# B&R Automation Studio project NAINV104C00R8L515F00 (part 28)

#### Act_Background_RequestedBoardChk.st
```iecst
(** 2023-04-11 **)
ACTION Act_Background_RequestedBoardChk:

	IF eStatus2 <> Error  THEN
		bBoardChkReq := FALSE;
		memset(ADR(tyBoardAvailableReq),0,SIZEOF(tyBoardAvailableReq));
		IF bProcessBoardForecastId AND bNotAvlNotRdy  THEN //process boardforecast
			tyBoardAvailableReq.tyAvl.bProductTypeId	 		:= tyBoardForecastAcc.tyAvl.bProductTypeId;
			tyBoardAvailableReq.tyData.sProductTypeId 			:= tyBoardForecastAcc.tyData.sProductTypeId	;
			tyBoardAvailableReq.tyAvl.bThickness 				:= tyBoardForecastAcc.tyAvl.bThickness;
			tyBoardAvailableReq.tyAvl.bWidth 					:= tyBoardForecastAcc.tyAvl.bWidth;
			tyBoardAvailableReq.tyData.rWidth 					:= tyBoardForecastAcc.tyData.rWidth;
			tyBoardAvailableReq.tyAvl.bTopClearanceHeight 		:= tyBoardForecastAcc.tyAvl.bTopClearanceHeight;
			tyBoardAvailableReq.tyAvl.bBottomClearanceHeight 	:= tyBoardForecastAcc.tyAvl.bBottomClearanceHeight;
			tyBoardAvailableReq.tyData.eFlippedBoard 			:= tyBoardForecastAcc.tyData.eFlippedBoard;
			tyBoardAvailableReq.tyData.rThickness 				:= tyBoardForecastAcc.tyData.rThickness;
			tyBoardAvailableReq.tyData.rTopClearanceHeight 		:= tyBoardForecastAcc.tyData.rTopClearanceHeight;
			tyBoardAvailableReq.tyData.rBottomClearanceHeight 	:= tyBoardForecastAcc.tyData.rBottomClearanceHeight;
			bBoardChkReq := TRUE;
		ELSIF  bRcvBoardInfoOk AND bManuallInsertLastZone THEN //process query board info
			tyBoardAvailableReq.tyAvl.bProductTypeId	 		:= tySendBoardInfoAcc.tyAvl.bProductTypeId;
			tyBoardAvailableReq.tyData.sProductTypeId 			:= tySendBoardInfoAcc.tyData.sProductTypeId;
			tyBoardAvailableReq.tyAvl.bThickness 				:= tySendBoardInfoAcc.tyAvl.bThickness;
			tyBoardAvailableReq.tyAvl.bWidth 					:= tySendBoardInfoAcc.tyAvl.bWidth;
			tyBoardAvailableReq.tyData.rWidth 					:= tySendBoardInfoAcc.tyData.rWidth;
			tyBoardAvailableReq.tyAvl.bTopClearanceHeight 		:= tySendBoardInfoAcc.tyAvl.bTopClearanceHeight;
			tyBoardAvailableReq.tyAvl.bBottomClearanceHeight 	:= tySendBoardInfoAcc.tyAvl.bBottomClearanceHeight;
			tyBoardAvailableReq.tyData.eFlippedBoard 			:= tySendBoardInfoAcc.tyData.eFlippedBoard;
			tyBoardAvailableReq.tyData.rThickness 				:= tySendBoardInfoAcc.tyData.rThickness;
			tyBoardAvailableReq.tyData.rTopClearanceHeight 		:= tySendBoardInfoAcc.tyData.rTopClearanceHeight;
			tyBoardAvailableReq.tyData.rBottomClearanceHeight 	:= tySendBoardInfoAcc.tyData.rBottomClearanceHeight;
			bBoardChkReq := TRUE;
		ELSIF p_bAccDataRdy THEN
			memcpy(ADR(tyBoardAvailableReq),ADR(tyBoardAvailableRcv),SIZEOF(tyBoardAvailableRcv));
			bBoardChkReq := TRUE;
		END_IF
		//ADD
		IF bBoardChkReq AND (bTransporting = FALSE) AND (p_bOpsRun = TRUE) THEN

			bAccDataReq		:= FALSE;
			bBABlkUS		:= FALSE;
			bOverWriteSlt	:= FALSE;
			bOverWriteWidth	:= FALSE;

			IF p_tyParam.bCmpTypeId = TRUE THEN	//"Compare Type ID" Ticked

				IF tyBoardAvailableReq.tyAvl.bProductTypeId = TRUE THEN	//Check if there is Product Type Id in B.A msg

					IF tyBoardAvailableReq.tyData.sProductTypeId <> p_sRecipeNm THEN	//Product Type Id Different

						bAccDataReq	    := TRUE;	//Require To Load New Recipe
						bBABlkUS		:= TRUE;

						sReqRecipeNm	:= tyBoardAvailableReq.tyData.sProductTypeId;
						diReqWidthInUM	:= REAL_TO_DINT(tyBoardAvailableReq.tyData.rWidth * 1000);

					ELSE	//Product Type Id Same (After accepted or Originally same)

						IF p_tyParam.bCmpParam = TRUE THEN	//"Compare Param" Ticked
							IF tyBoardAvailableReq.tyAvl.bThickness AND tyBoardAvailableReq.tyAvl.bTopClearanceHeight AND tyBoardAvailableReq.tyAvl.bBottomClearanceHeight AND p_bBASltEn THEN	//Camparing Slot Parameters if p_bBASltEn = TRUE
								udiStatus2	:= fHermesCmpSlt(tyBoardAvailableReq.tyData.eFlippedBoard , tyBoardAvailableReq.tyData.rThickness , tyBoardAvailableReq.tyData.rTopClearanceHeight , tyBoardAvailableReq.tyData.rBottomClearanceHeight , p_diMinSltValue , p_diMaxSltValue , p_diPitch , p_diSltToSltInUM , p_diTtlSlt);

								IF udiStatus2 <> 0 THEN

									bBABlkUS	:= TRUE;

									eStatus2	:= Error;

									IF udiStatus2 = 2914 THEN
										udiStatus2	:= 10108;	//Input First Slot Is Invalid
									ELSIF udiStatus2 = 2915 THEN
										udiStatus2	:= 10109;	//Input Last Slot Is Invalid
									ELSIF udiStatus2 = 2916 THEN
										udiStatus2	:= 10110;	//Input Pitch Is Invalid
									ELSIF udiStatus2 = 2917 THEN
										udiStatus2	:= 10111;	//Input Slot To Slot Distance Is Invalid
									ELSIF udiStatus2 = 2918 THEN
										udiStatus2	:= 10112;	//Input Total Slot Is Invalid
									ELSIF udiStatus2 = 2919 THEN
										udiStatus2	:= 10113;	//Input Thickness Is Invalid
									ELSIF udiStatus2 = 2920 THEN
										udiStatus2	:= 10114;	//Input Top Clearance Height Is Invalid
									ELSIF udiStatus2 = 2921 THEN
										udiStatus2	:= 10115;	//Input Bottom Clearance Height Is Invalid
									ELSIF udiStatus2 = 2922 THEN
										udiStatus2	:= 10116;	//Recipe First Slot Value & Board Available Data Not Match With Same Product Type Id
									ELSIF udiStatus2 = 2923 THEN
										udiStatus2	:= 10117;	//Recipe Last Slot Value & Board Available Data Not Match With Same Product Type Id
									ELSIF udiStatus2 = 2924 THEN
										udiStatus2	:= 10118;	//Recipe Pitch Value & Board Available Data Not Match With Same Product Type Id
									END_IF

									fHermesAddOneMsgSend(ADR(a_eMsgSend) , ADR(udiMsgSendBffr) , HermesMsgTypeNotification);

									tyNotificationSnd.tyAvl.bSeverity			:= TRUE;
									tyNotificationSnd.tyAvl.bNotificationCode	:= TRUE;
									tyNotificationSnd.tyAvl.bDescription		:= TRUE;
									tyNotificationSnd.tyData.eSeverity			:= HermesSeverityError;
									tyNotificationSnd.tyData.iNotificationCode	:= UDINT_TO_INT(udiStatus2);
									tyNotificationSnd.tyData.sDescription		:= a_tyAlmText[udiStatus2].sAlmText;

								END_IF
							END_IF

							IF tyBoardAvailableReq.tyAvl.bWidth AND p_bBAWidthEn THEN	//Comparing Width Parameter if p_bBAWidthEn = TRUE
								IF REAL_TO_DINT(tyBoardAvailableReq.tyData.rWidth * 1000) <> p_diWidthInUM THEN

									bBABlkUS	:= TRUE;

									eStatus2	:= Error;
									udiStatus2	:= 10119;	//Width Different With Same Product Type Id

									fHermesAddOneMsgSend(ADR(a_eMsgSend) , ADR(udiMsgSendBffr) , HermesMsgTypeNotification);

									tyNotificationSnd.tyAvl.bSeverity			:= TRUE;
									tyNotificationSnd.tyAvl.bNotificationCode	:= TRUE;
									tyNotificationSnd.tyAvl.bDescription		:= TRUE;
									tyNotificationSnd.tyData.eSeverity			:= HermesSeverityError;
									tyNotificationSnd.tyData.iNotificationCode	:= UDINT_TO_INT(udiStatus2);
									tyNotificationSnd.tyData.sDescription		:= a_tyAlmText[udiStatus2].sAlmText;

								END_IF
							END_IF

						END_IF

					END_IF

				ELSE

					eStatus2	:= Error;
					udiStatus2	:= 10158;	//Product Type Id Not Receive From Upstream

					fHermesAddOneMsgSend(ADR(a_eMsgSend) , ADR(udiMsgSendBffr) , HermesMsgTypeNotification);

					tyNotificationSnd.tyAvl.bSeverity			:= TRUE;
					tyNotificationSnd.tyAvl.bNotificationCode	:= TRUE;
					tyNotificationSnd.tyAvl.bDescription		:= TRUE;
					tyNotificationSnd.tyData.eSeverity			:= HermesSeverityError;
					tyNotificationSnd.tyData.iNotificationCode	:= UDINT_TO_INT(udiStatus2);
					tyNotificationSnd.tyData.sDescription		:= a_tyAlmText[udiStatus2].sAlmText;

				END_IF

			ELSE	//"Compare Type ID" Not Ticked

				IF p_tyParam.bOverwrite THEN	//"Overwrite" Ticked

					IF tyBoardAvailableReq.tyAvl.bThickness AND tyBoardAvailableReq.tyAvl.bTopClearanceHeight AND tyBoardAvailableReq.tyAvl.bBottomClearanceHeight AND p_bBASltEn THEN	//Camparing Slot Parameters

						udiStatus2	:= fHermesCmpSlt(tyBoardAvailableReq.tyData.eFlippedBoard , tyBoardAvailableReq.tyData.rThickness , tyBoardAvailableReq.tyData.rTopClearanceHeight , tyBoardAvailableReq.tyData.rBottomClearanceHeight , p_diMinSltValue , p_diMaxSltValue , p_diPitch , p_diSltToSltInUM , p_diTtlSlt);

						IF udiStatus2 <> 0 THEN

							bAccDataReq		:= TRUE;
							bBABlkUS			:= TRUE;
							bOverWriteSlt	:= TRUE;

							fbGetSlt.eFlippedBrd				:= tyBoardAvailableReq.tyData.eFlippedBoard;
							fbGetSlt.rThicknessInMM				:= tyBoardAvailableReq.tyData.rThickness;
							fbGetSlt.rTopClearanceHeightInMM	:= tyBoardAvailableReq.tyData.rTopClearanceHeight;
							fbGetSlt.rBtmClearanceHeightInMM	:= tyBoardAvailableReq.tyData.rBottomClearanceHeight;
							fbGetSlt.diSltToSltInUM				:= p_diSltToSltInUM;
							fbGetSlt.diTtlSlt					:= p_diTtlSlt;
							fbGetSlt;

							diReqMinSltValue	:= fbGetSlt.diMinSltValue;
							diReqMaxSltValue	:= fbGetSlt.diMaxSltValue;
							diReqPitch			:= fbGetSlt.diPitch;

						END_IF

					END_IF

					IF tyBoardAvailableReq.tyAvl.bWidth  AND p_bBAWidthEn (*AND p_usiLinkProdRcpCurrRcpMcMod = 0*) THEN	//Comparing Width Parameter
						IF REAL_TO_DINT(tyBoardAvailableReq.tyData.rWidth * 1000) <> p_diWidthInUM THEN

							bAccDataReq		:= TRUE;
							bBABlkUS			:= TRUE;
							bOverWriteWidth	:= TRUE;

							diReqWidthInUM	:= REAL_TO_DINT(tyBoardAvailableReq.tyData.rWidth * 1000);

						END_IF
					END_IF

				ELSE	//"Compare Type ID" Not Ticked and "Overwrite" Not Ticked, Error if not same

					IF tyBoardAvailableReq.tyAvl.bThickness AND tyBoardAvailableReq.tyAvl.bTopClearanceHeight AND tyBoardAvailableReq.tyAvl.bBottomClearanceHeight AND p_bBASltEn AND p_bRdyRcv THEN	//Camparing Slot Parameters
						udiStatus2	:= fHermesCmpSlt(tyBoardAvailableReq.tyData.eFlippedBoard , tyBoardAvailableReq.tyData.rThickness , tyBoardAvailableReq.tyData.rTopClearanceHeight , tyBoardAvailableReq.tyData.rBottomClearanceHeight , p_diMinSltValue , p_diMaxSltValue , p_diPitch , p_diSltToSltInUM , p_diTtlSlt);

						IF udiStatus2 <> 0 THEN

							bBABlkUS		:= TRUE;

							eStatus2	:= Error;

							IF udiStatus2 = 2914 THEN
								udiStatus2	:= 10120;	//Input First Slot Is Invalid
							ELSIF udiStatus2 = 2915 THEN
								udiStatus2	:= 10121;	//Input Last Slot Is Invalid
							ELSIF udiStatus2 = 2916 THEN
								udiStatus2	:= 10122;	//Input Pitch Is Invalid
							ELSIF udiStatus2 = 2917 THEN
								udiStatus2	:= 10123;	//Input Slot To Slot Distance Is Invalid
							ELSIF udiStatus2 = 2918 THEN
								udiStatus2	:= 10124;	//Input Total Slot Is Invalid
							ELSIF udiStatus2 = 2919 THEN
								udiStatus2	:= 10125;	//Input Thickness Is Invalid
							ELSIF udiStatus2 = 2920 THEN
								udiStatus2	:= 10126;	//Input Top Clearance Height Is Invalid
							ELSIF udiStatus2 = 2921 THEN
								udiStatus2	:= 10127;	//Input Bottom Clearance Height Is Invalid
							ELSIF udiStatus2 = 2922 THEN
								udiStatus2	:= 10128;	//Recipe First Slot Value & Board Available Data Not Match With Same Product Type Id
							ELSIF udiStatus2 = 2923 THEN
								udiStatus2	:= 10129;	//Recipe Last Slot Value & Board Available Data Not Match With Same Product Type Id
							ELSIF udiStatus2 = 2924 THEN
								udiStatus2	:= 10130;	//Recipe Pitch Value & Board Available Data Not Match With Same Product Type Id
							END_IF

							fHermesAddOneMsgSend(ADR(a_eMsgSend) , ADR(udiMsgSendBffr) , HermesMsgTypeNotification);

							tyNotificationSnd.tyAvl.bSeverity			:= TRUE;
							tyNotificationSnd.tyAvl.bNotificationCode	:= TRUE;
							tyNotificationSnd.tyAvl.bDescription		:= TRUE;
							tyNotificationSnd.tyData.eSeverity			:= HermesSeverityError;
							tyNotificationSnd.tyData.iNotificationCode	:= UDINT_TO_INT(udiStatus2);
							tyNotificationSnd.tyData.sDescription		:= a_tyAlmText[udiStatus2].sAlmText;

						END_IF
					END_IF

					IF tyBoardAvailableReq.tyAvl.bWidth AND p_bBAWidthEn AND p_bRdyRcv THEN	//Comparing Width Parameter
						IF REAL_TO_DINT(tyBoardAvailableReq.tyData.rWidth * 1000) <> p_diWidthInUM THEN

							bBABlkUS		:= TRUE;

							eStatus2	:= Error;
							udiStatus2	:= 10131;	//Width Different With Same Product Type Id

							fHermesAddOneMsgSend(ADR(a_eMsgSend) , ADR(udiMsgSendBffr) , HermesMsgTypeNotification);

							tyNotificationSnd.tyAvl.bSeverity			:= TRUE;
							tyNotificationSnd.tyAvl.bNotificationCode	:= TRUE;
							tyNotificationSnd.tyAvl.bDescription		:= TRUE;
							tyNotificationSnd.tyData.eSeverity			:= HermesSeverityError;
							tyNotificationSnd.tyData.iNotificationCode	:= UDINT_TO_INT(udiStatus2);
							tyNotificationSnd.tyData.sDescription		:= a_tyAlmText[udiStatus2].sAlmText;

						END_IF
					END_IF

				END_IF

			END_IF
			                                                       //Add
		ELSIF NOT(bBoardChkReq) OR bTransporting = TRUE THEN //AND p_bUIInsertBrdPrep = FALSE THEN

			bAccDataReq		:= FALSE;
			bBABlkUS		:= FALSE;
			bOverWriteSlt	:= FALSE;
			bOverWriteWidth	:= FALSE;

		END_IF

		//reset bProcessBoardForecastId
		IF bProcessBoardForecastId = TRUE AND bBoardChkReq AND (bTransporting = FALSE) AND (p_bOpsRun = TRUE) THEN //reset condition
			IF bBABlkUS = FALSE OR  (bBFBlkUS AND eStatus2 = Error) THEN
				IF eStatus2 <> Error THEN
					bReplyMcRdyId := TRUE;
				END_IF
				bProcessBoardForecastId := FALSE;
			END_IF
		END_IF

	ELSE

		bAccDataReq		:= FALSE;
		bBABlkUS		:= TRUE;
		bOverWriteSlt	:= FALSE;
		bOverWriteWidth	:= FALSE;
		bBoardChkReq  := FALSE;
	END_IF

END_ACTION
```

#### Act_Background_Route.st
```iecst
(** 2021-08-01 **)
ACTION Act_Background_Route:

	//US Routing function

	//iGotoLane 0 Default Lane
	//iGotoLane 1 Route1
	IF NOT(p_bProcessRouteEn) THEN
		bReverseDSSndBfWBrdID := FALSE;
		bManualRmvBrdCond := FALSE;
		iGotoLane	:= 0;
		bProcessRouteReversal := FALSE;
		bTriggerRouteReversal := FALSE;
	ELSE
		// reversal condition
		IF EDGEPOS(tyBoardAvailableRcv.tyData.iRoute  = 900 AND tyBoardAvailableRcv.tyAvl.bRoute) THEN //flipping station reversal condition
			tyBoardAvailableRcv.tyAvl.bRoute := FALSE;
			bProcessRouteReversal := TRUE;
		ELSIF EDGEPOS(tyBoardAvailableRcv.tyAvl.bFlippedBoard  AND tyBoardAvailableRcv.tyData.eFlippedBoard = HermesFlippedBoardTopSideUp) THEN
			bTriggerRouteReversal := TRUE;
		END_IF

		//receiving Route
		IF	NOT(tyBoardAvailableRcv.tyAvl.bRoute)   THEN
			iGotoLane := 0; //default, depend on priority
		ELSE
			IF  p_bManualRmvRoute AND tyBoardAvailableRcv.tyData.iRoute  = 999  THEN
				bManualRmvBrdCond := TRUE;

			ELSIF p_bReturnRoute AND (
				(bProcessRouteReversal AND bProcessRouteMachine
				OR
				bTriggerRouteReversal AND bTriggerRouteMachine)
				OR bReverseDSSndBfWBrdID) THEN
				IF bProcessRouteReversal  THEN //Route Guide (900),flipper as downstream
					bReverseDSSndBfWBrdID := TRUE;
					bTriggerUpdateRoute  := FALSE;
					bProcessRouteReversal := FALSE;
				ELSIF bTriggerRouteReversal THEN //process as downstream
					bReverseDSSndBfWBrdID := TRUE;
					bTriggerUpdateRoute  := TRUE;
					bTriggerRouteReversal := FALSE;
				END_IF

				//Reset
				fbRstReverseDSSndBF(IN:= bReverseDSSndBfWBrdID AND NOT(p_bReceiveReverseUSMcRdy));
				IF (bReverseDSSndBfWBrdID AND p_bReceiveReverseUSMcRdy) OR fbRstReverseDSSndBF.Q THEN
					bReverseDSSndBfWBrdID := FALSE;
					bTriggerUpdateRoute := FALSE;
				END_IF
			ELSIF p_bNomRouteEn THEN
				iMinDis := 0;
				FOR usidx := 0 TO 2 DO
					//bChecking Closest Route
					IF tyBoardAvailableRcv.tyData.iRoute = pa_tyHermesDSParam[usidx].iLaneID THEN
						iGotoLane := usidx; //iGotoLane switch direction
						EXIT;
					ELSIF iMinDis = 0 THEN
						iMinDis := ABS(tyBoardAvailableRcv.tyData.iRoute - pa_tyHermesDSParam[usidx].iLaneID);
						iGotoLane := usidx;
					ELSE
						IF iMinDis > ABS(tyBoardAvailableRcv.tyData.iRoute - pa_tyHermesDSParam[usidx].iLaneID) THEN
							iGotoLane := usidx;
							iMinDis := ABS(tyBoardAvailableRcv.tyData.iRoute - pa_tyHermesDSParam[usidx].iLaneID);
						END_IF
					END_IF
				END_FOR
			END_IF
		END_IF

		//Process 900
		//when to reset block DS signal

		//Process 999
		//fbRstReverseDSSndBF(IN:= bManualRmvBrdCond);

	//	bBlkUS := bBlkUS OR bReverseDSSndBfWBrdID; //OR p_bSwitchtoReverseReceive;
	END_IF

	//reverse route, input receiving
	IF NOT(p_bReverseReceiveRoute) THEN
		bSwitchtoReverseReceive := FALSE;
	ELSE
		//process Reverse Input
		IF bSwitchtoReverseReceive = FALSE  AND EDGEPOS(p_tyDSHermesCurrBASnd.tyData.sBoardId = tyBoardForecastRcv.tyData.sBoardId AND tyBoardForecastRcv.tyData.sBoardId <> '' AND tyBoardForecastRcv.tyAvl.bBoardId) THEN
			tyBoardForecastRcv.tyAvl.bBoardId := FALSE;
			bSwitchtoReverseReceive := TRUE; //when to reset ReverseRcv back , if the BASnd not the same anymore
		ELSIF bSwitchtoReverseReceive = TRUE
			AND (EDGEPOS(tyMsgTypeRcv.bTransportFinished AND tyTransportFinished.tyData.eTransferState = HermesTransferStateComplete )
			OR EDGEPOS(tyMsgTypeRcv.bBoardForecast AND tyBoardForecastRcv.tyData.sBoardId = ''  )) THEN
			tyBoardForecastRcv.tyAvl.bBoardId := FALSE;
			bSwitchtoReverseReceive := FALSE;
		END_IF
		fbRstReverseRcvGate(IN:= bSwitchtoReverseReceive);
		bNotifyRstReverseRcvGate := fbRstReverseRcvGate.Q;
		//	bBlkUS := bBlkUS OR NOT(bSwitchtoReverseReceive);

		bReverseRcvBlkUS := NOT(bSwitchtoReverseReceive);
	END_IF

	//bBlkUS := bBlkUS OR p_bUSHermes2SwitchtoReverseRcv;
END_ACTION
```

#### Act_Background_Sequence.st
```iecst
 (** 2019-05-04 **)
ACTION Act_Background_Sequence:

	IF eStatus1 <> Error THEN

		IF p_bOpsRun = FALSE THEN
			p_bRcvIncompl	:= TRUE;
		END_IF

		IF tyMsgTypeRcv.bTransportFinished = TRUE THEN
			IF tyTransportFinished.tyData.eTransferState = HermesTransferStateNotStarted THEN
				p_bRcvNotStart	:= TRUE;
			ELSIF tyTransportFinished.tyData.eTransferState = HermesTransferStateIncomplete THEN
				p_bRcvIncompl	:= TRUE;
			END_IF
		END_IF

		bBlkUS := bBABlkUS OR  bBFBlkUS OR bManuallInsertLastZone
			OR bReverseDSSndBfWBrdID
			OR bReverseRcvBlkUS
			OR NOT(p_bHermesSwitchtoRvrseTransport); //no for reversal gate

		bBoardAvailableRcved := tyMsgTypeRcv.bBoardAvailable;

		//Sequence
		fbSequenceUS.bRstState		:= bRstState;
		fbSequenceUS.bRdyRcv		:= (p_bRdyRcv) AND (eStatus2 <> Error);
		fbSequenceUS.bBlkUS			:= bBlkUS;
		fbSequenceUS.bRdyTransport	:= p_bRdyTransport;
		fbSequenceUS.bRcvCompl		:= p_bRcvCompl;
		fbSequenceUS.bRcvIncompl	:= p_bRcvIncompl;
		fbSequenceUS.bRcvNotStart	:= p_bRcvNotStart;
		fbSequenceUS.bProcessBoardForecastId     	:= bProcessBoardForecastId; //Received BoardForecastId

		fbSequenceUS(bEn := TRUE);

		bNotAvlNotRdy                               := fbSequenceUS.bNotAvlNotRdy;

		bUSRdy		                               	:= fbSequenceUS.bUSRdy; //bUSRdy:= (eState = HermesStateBoardAvailable) OR (eState = HermesStateAvailableAndReady) OR (eState >= HermesStateTransporting);
		bDSRdy		                               	:= fbSequenceUS.bDSRdy;
		bTransporting                             	:= fbSequenceUS.bTransporting;
		bStopTransport                            	:= fbSequenceUS.bStopTransport;
		bUSGdRdy                                   	:= (tyBoardAvailableRcv.tyAvl.bFailedBoard = FALSE) OR ((tyBoardAvailableRcv.tyAvl.bFailedBoard = TRUE) AND (tyBoardAvailableRcv.tyData.eFailedBoard <> HermesFailedBoard));
		bDSGdRdy                                   	:= (tyMachineReady.tyAvl.bFailedBoard = FALSE) OR ((tyMachineReady.tyAvl.bFailedBoard = TRUE) AND (tyMachineReady.tyData.eFailedBoard <> HermesFailedBoard));

		//Action (defined 1 as bypass, 2 as flip)
		iAction										:= (tyBoardAvailableRcv.tyAvl.bAction = TRUE)*(tyBoardAvailableRcv.tyData.iAction);

		IF fbSequenceUS.eState >= HermesStateNotAvailableNotReady THEN
			bHandshakeDone	:= TRUE;
		ELSE
			bHandshakeDone	:= FALSE;
		END_IF

		IF EDGEPOS(fbSequenceUS.eState = HermesStateTransporting) THEN
			p_bRcvCompl		:= FALSE;
			p_bRcvIncompl	:= FALSE;
			p_bRcvNotStart	:= FALSE;
		END_IF

		IF fbSequenceUS.eMsgTypeSnd = HermesMsgTypeServiceDescription THEN
			fHermesAddOneMsgSend(ADR(a_eMsgSend) , ADR(udiMsgSendBffr) , HermesMsgTypeServiceDescription);

			tyServiceDescriptionSnd.tyData.sMachineId                                       := p_sMcId;
			tyServiceDescriptionSnd.tyData.iLaneId											:= p_tyParam.iLaneID;
			tyServiceDescriptionSnd.tyData.sInterfaceId										:= p_tyParam.sUpstreamInterfaceId;
			tyServiceDescriptionSnd.tyData.sVersion											:= p_sVersion;
			tyServiceDescriptionSnd.tyData.tySupportedFeatures.bFeatureCheckAliveResponse	:= (p_tyParam.bFeatureCheckAliveResponse) AND (p_tyParam.tRcvAlive <> T#0s) AND (p_tyParam.tSndAlive <> T#0s);
			tyServiceDescriptionSnd.tyData.tySupportedFeatures.bFeatureBoardForecast		:= p_tyParam.bFeatureBoardForecast;
			tyServiceDescriptionSnd.tyData.tySupportedFeatures.bFeatureQueryBoardInfo		:= p_tyParam.bFeatureQueryBoardInfo;
			tyServiceDescriptionSnd.tyData.tySupportedFeatures.bFeatureSendBoardInfo		:= FALSE;

			tyServiceDescriptionSnd.tyAvl.bMachineId										:= TRUE;
			tyServiceDescriptionSnd.tyAvl.bLaneId											:= tyServiceDescriptionSnd.tyData.iLaneId <> 0;
			tyServiceDescriptionSnd.tyAvl.bInterfaceId										:= tyServiceDescriptionSnd.tyData.sInterfaceId <> '';
			tyServiceDescriptionSnd.tyAvl.bVersion											:= TRUE;
			tyServiceDescriptionSnd.tyAvl.bSupportedFeatures								:= p_tyParam.bFeatureCheckAliveResponse OR p_tyParam.bFeatureBoardForecast OR p_tyParam.bFeatureQueryBoardInfo;
			tyServiceDescriptionSnd.tyAvl.tySupportedFeatures.bFeatureCheckAliveResponse	:= (p_tyParam.bFeatureCheckAliveResponse) AND (p_tyParam.tRcvAlive <> T#0s) AND (p_tyParam.tSndAlive <> T#0s);
			tyServiceDescriptionSnd.tyAvl.tySupportedFeatures.bFeatureBoardForecast			:= p_tyParam.bFeatureBoardForecast;
			tyServiceDescriptionSnd.tyAvl.tySupportedFeatures.bFeatureQueryBoardInfo		:= p_tyParam.bFeatureQueryBoardInfo;
			tyServiceDescriptionSnd.tyAvl.tySupportedFeatures.bFeatureSendBoardInfo			:= FALSE;

		ELSIF fbSequenceUS.eMsgTypeSnd = HermesMsgTypeMachineReady THEN
			IF bReplyMcRdyId = FALSE THEN

			    fHermesAddOneMsgSend(ADR(a_eMsgSend) , ADR(udiMsgSendBffr) , HermesMsgTypeMachineReady);

		    	tyMachineReady.tyData.eFailedBoard			:= p_eFailedBoard;
				tyMachineReady.tyAvl.bFailedBoard			:= TRUE;
			    tyMachineReady.tyAvl.bForecastId			:= FALSE;
				tyMachineReady.tyAvl.bBoardId				:= FALSE;
			    tyMachineReady.tyAvl.bProductTypeId			:= FALSE;
			    tyMachineReady.tyAvl.bFlippedBoard			:= FALSE;
			    tyMachineReady.tyAvl.bLength				:= FALSE;
			    tyMachineReady.tyAvl.bWidth					:= FALSE;
			    tyMachineReady.tyAvl.bThickness				:= FALSE;
			    tyMachineReady.tyAvl.bConveyorSpeed			:= FALSE;
			    tyMachineReady.tyAvl.bTopClearanceHeight	:= FALSE;
			    tyMachineReady.tyAvl.bBottomClearanceHeight	:= FALSE;
		    	tyMachineReady.tyAvl.bWeight				:= FALSE;
				tyMachineReady.tyAvl.bWorkOrderId			:= FALSE;
				tyMachineReady.tyAvl.bBatchId    			:= FALSE;

			ELSE
				fHermesAddOneMsgSend(ADR(a_eMsgSend) , ADR(udiMsgSendBffr) , HermesMsgTypeMachineReady);

				tyMachineReady.tyData.eFailedBoard			:= p_eFailedBoard;
				tyMachineReady.tyData.sForecastId	        := tyBoardForecastAcc.tyData.sForecastId;
				tyMachineReady.tyData.sProductTypeId	    := p_sRecipeNm;
				tyMachineReady.tyData.rWidth	            := DINT_TO_REAL(p_diWidthInUM) / 1000;
				tyMachineReady.tyAvl.bFailedBoard			:= TRUE;
				tyMachineReady.tyAvl.bForecastId			:= tyBoardForecastAcc.tyData.sForecastId<>'';
				tyMachineReady.tyAvl.bBoardId				:= FALSE;
				tyMachineReady.tyAvl.bProductTypeId			:= tyBoardForecastAcc.tyData.sProductTypeId<>'';
				tyMachineReady.tyAvl.bFlippedBoard			:= FALSE;
				tyMachineReady.tyAvl.bLength				:= FALSE;
				tyMachineReady.tyAvl.bWidth					:= tyMachineReady.tyData.rWidth<>0;
				tyMachineReady.tyAvl.bThickness				:= FALSE;
				tyMachineReady.tyAvl.bConveyorSpeed			:= FALSE;
				tyMachineReady.tyAvl.bTopClearanceHeight	:= FALSE;
				tyMachineReady.tyAvl.bBottomClearanceHeight	:= FALSE;
				tyMachineReady.tyAvl.bWeight				:= FALSE;
				tyMachineReady.tyAvl.bWorkOrderId			:= FALSE;
				tyMachineReady.tyAvl.bBatchId		    	:= FALSE;

			END_IF

		ELSIF fbSequenceUS.eMsgTypeSnd = HermesMsgTypeRevokeMachineReady THEN
			fHermesAddOneMsgSend(ADR(a_eMsgSend) , ADR(udiMsgSendBffr) , HermesMsgTypeRevokeMachineReady);

		ELSIF fbSequenceUS.eMsgTypeSnd = HermesMsgTypeStartTransport THEN
			fHermesAddOneMsgSend(ADR(a_eMsgSend) , ADR(udiMsgSendBffr) , HermesMsgTypeStartTransport);

			tyStartTransport.tyData.sBoardId		:= tyBoardAvailableRcv.tyData.sBoardId;

			tyStartTransport.tyAvl.bBoardId			:= TRUE;
			tyStartTransport.tyAvl.bConveyorSpeed	:= FALSE;

		ELSIF fbSequenceUS.eMsgTypeSnd = HermesMsgTypeStopTransport THEN
			fHermesAddOneMsgSend(ADR(a_eMsgSend) , ADR(udiMsgSendBffr) , HermesMsgTypeStopTransport);

			IF p_bRcvCompl = TRUE THEN
				tyStopTransport.tyData.eTransferState	:= HermesTransferStateComplete;
			ELSIF p_bRcvIncompl = TRUE THEN
				tyStopTransport.tyData.eTransferState	:= HermesTransferStateIncomplete;
			ELSE
				tyStopTransport.tyData.eTransferState	:= HermesTransferStateNotStarted;
			END_IF
			tyStopTransport.tyData.sBoardId				:= tyStartTransport.tyData.sBoardId;

			tyStopTransport.tyAvl.bTransferState		:= TRUE;
			tyStopTransport.tyAvl.bBoardId				:= TRUE;

		END_IF

	END_IF

	bStopTransportSent := fbSequenceUS.eMsgTypeSnd = HermesMsgTypeStopTransport;

END_ACTION
```

#### Act_Background_Stop.st
```iecst
(** 2019-03-15 **)
ACTION Act_Background_Stop:

	IF EDGEPOS(bStop) THEN

		fHermesAddOneMsgSend(ADR(a_eMsgSend) , ADR(udiMsgSendBffr) , HermesMsgTypeNotification);

		tyNotificationSnd.tyAvl.bSeverity			:= TRUE;
		tyNotificationSnd.tyAvl.bNotificationCode	:= TRUE;
		tyNotificationSnd.tyAvl.bDescription		:= TRUE;
		tyNotificationSnd.tyData.eSeverity			:= HermesSeverityInfo;
		tyNotificationSnd.tyData.iNotificationCode	:= 5;
		tyNotificationSnd.tyData.sDescription		:= 'Machine Shutdown';

	END_IF

	IF bStop = TRUE THEN

		IF a_eMsgSend[0] = HermesMsgTypeNA THEN

			bRstConnection	:= TRUE;

			IF udiTCPIdent = 0 THEN

				bRun	:= FALSE;

			END_IF

		END_IF

	END_IF

END_ACTION
```

#### Act_Background_TCPClose.st
```iecst
(** 2019-06-10 **)
ACTION Act_Background_TCPClose:

	//Close TCP Connection
	IF p_bInternalUse = FALSE THEN
		fbClose.udiTCPIdent	:= udiTCPIdent;
		fbClose(bEn := TRUE);

		IF fbClose.udiStatus = 0 THEN
			udiTCPIdent	:= 0;
			fbClose(bEn := FALSE);

		ELSIF fbClose.udiStatus < 65534 THEN
			udiTCPIdent	:= 0;
			eStatus1	:= Error;

			IF fbClose.udiStatus = 2300 THEN
				udiStatus1	:= 10146;	//Invalid Ident While Closing TCP
			ELSIF fbClose.udiStatus = 2310 THEN
				udiStatus1	:= 10147;	//Closing TCP Error
			ELSE
				udiStatus1	:= fbClose.udiStatus;
			END_IF

		END_IF

	ELSE
		udiTCPIdent	:= 0;

	END_IF

END_ACTION
```

#### Act_CombineErr.st
```iecst
(** 2019-03-15 **)
ACTION Act_CombineErr:

	//Combine Error
	IF eStatus = Error OR eStatus1 = Error OR eStatus2 = Error OR eStatus3 = Error OR eStatus4 = Error THEN
		eMainStatus	:= Error;
	ELSE
		eMainStatus	:= eStatus;
	END_IF

END_ACTION
```

#### Act_InitGlobal.st
```iecst
(** 2019-06-28 **)
ACTION Act_InitGlobal:

	(* Always Change If Project Change *)

	//Pass Data To Link
	p_bLinkStartupRun ACCESS p_StartupRun;
	p_eLinkMcParamUSCommMod ACCESS p_McParamUSComm2Mod;

	p_eLinkConvDir ACCESS p_NtParamProjConvDir;
	p_bLinkDILeftSen ACCESS p_DIConvLftSen;
	p_bLinkDIRightSen ACCESS p_DIConvRgtSen;

	p_bLinkOpsInvertStepInitDone ACCESS p_OpsInvertStepInitDone;
	p_bLinkOpsRun ACCESS p_OpsRun;

	//Pass Data To Internal Use
	p_udiRstErr ACCESS p_RstErrReset;
	p_bPrep ACCESS p_NtParamHermesPrep;
	p_tyParam ACCESS p_HermesUSParam2;
	p_sIPAddr ACCESS p_HWInfoIPAddr;
	p_tyDTStructure ACCESS p_TimeCurrDTStruct;
	p_dtCurrDT ACCESS p_TimeCurrDT;
	p_sMcId ACCESS p_McParamMcNm;
	p_sRecipeNm ACCESS p_ProdRcpCurrRcp0Nm;
	p_diWidthInUM ACCESS p_ProdRcpCurrRcp0Width;
	p_udiAliveIdleTimeInSec ACCESS p_NtParamUSHermes2AliveTmInSec;
	p_tConnTimeOut ACCESS p_NtParamUSHermes2ConnTO;
	p_diTransferInTO ACCESS p_McParamTranInErrDlyTm;
	p_bInterruptSen ACCESS p_DIConvLftSen;
	p_bOpsRun ACCESS p_OpsRun;
	p_udiFileKeepDay ACCESS p_NtParamUSHermes2FileKeepDay;
	p_sProgNm ACCESS p_NtParamUSHermes2ProgNm;
	p_bNtSettingsLoadDone ACCESS p_StartupNtSettingsLoadDone;
	p_bAccDataRdy ACCESS p_USHermes2USRdy;
	p_sRmtMcId ACCESS p_RmtHermesCurrentConfMcId;
	p_bRmtPrep ACCESS p_NtParamHermesRmtPrep;
	p_bRmtEn ACCESS p_McParamHermesRmtEn;
	pa_tyProdRcpList ACCESS p_ProdRcpCurrList;
	p_tyProdRcpCurrRcp ACCESS p_ProdRcpCurrRcp0;
	p_bMcParamMnlAccData ACCESS p_McParamMnlAccDat;
	p_bUIAccData ACCESS p_UIProdAccData;

	pa_tyHermesDSParam ACCESS pa_HermesDSParam;

	p_bHermesSwitchtoRvrseTransport ACCESS p_HermesSwitchtoReverseTransport;//;
	//Query Board Info
	p_bTransportFinished ACCESS p_DSHermesTransportFinish ;
	p_bQueryBoardInfo ACCESS p_UIQueryBoardInfo;
	p_bManualInsertZoneHvBrd ACCESS p_ConvHvBrd; //insert zone (can input conv or ouput conv)
	p_bManualInsertEndSen ACCESS p_DIConvRgtSen;
	p_bConvHvBrd ACCESS p_ConvHvBrd; //first zone
	//Reverse Machine Ready
	p_tyDSHermesCurrBASnd	ACCESS p_DSHermesBrdAvlSnd;
	(* Always Change If Project Change *)

END_ACTION
```

#### Act_Initial.st
```iecst
(** 2019-04-08 **)
ACTION Act_Initial:

	//Initial
	sStatTxt	:= a_sStatText[eStat];

	fbClntConnect.udiSndBffrSize		:= p_udiSndBffrSize;
	fbClntConnect.udiRcvBffrSize		:= p_udiRcvBffrSize;
	fbClntConnect.udiAliveIdleTmInSec	:= p_udiAliveIdleTimeInSec;
	fbClntConnect.tConnectTO			:= p_tConnTimeOut;
	fbClntConnect(bEn := FALSE);

	fbRcv.udiBffrSize	:= SIZEOF(sRcv);
	fbRcv.p_BffrDest	:= ADR(sRcv);
	fbRcv(bEn := FALSE);

	fbSend.p_BffrDest	:= ADR(sSnd);
	fbSend(bEn := FALSE);

	fbClose(bEn := FALSE);

	fbParseXMLTable.p_XMLTable	:= ADR(a_tyXMLTableDataRcv);

	fbCheckAlive(bEn := FALSE);

	fbCheckAliveSendPing(bEn := FALSE);

	fbCheckAliveRcvPing(bEn := FALSE);

	fbSequenceUS.p_tyMsgTypeRcv	:= ADR(tyMsgTypeRcv);
	fbSequenceUS(bEn := FALSE);

	fbSequenceTO(bEn := FALSE);

	fbFileAppend1.sDevice	:= 'Log';
	fbFileAppend1(bEn := FALSE);

	fbFileOldDel1.sDevice			:= 'Log';
	fbFileOldDel1.sPath				:= '';
	fbFileOldDel1.sKeyword			:= p_sProgNm;
	fbFileOldDel1.udiFileKeepDay	:= p_udiFileKeepDay;
	fbFileOldDel1(bEn := FALSE);

END_ACTION
```

#### Act_InitLocal.st
```iecst
(** 2019-06-28 **)
ACTION Act_InitLocal:

	//Input Reference Link To Local Variable
	p_eAct ACCESS ADR(eAct);
	p_udiRstErr ACCESS ADR(udiRstErr);
	p_bPrep ACCESS ADR(bPrep);
	p_bEn ACCESS ADR(bEn);
	p_bDis ACCESS ADR(bDis);
	p_tyParam ACCESS ADR(tyParam);
	p_sIPAddr ACCESS ADR(sIPAddr);
	p_tyDTStructure ACCESS ADR(tyDTStructure);
	p_dtCurrDT ACCESS ADR(dtCurrDT);
	p_bRdyRcv ACCESS ADR(bRdyRcv);
	p_bRdyTransport ACCESS ADR(bRdyTransport);
	p_bRcvCompl ACCESS ADR(bRcvCompl);
	p_bRcvIncompl ACCESS ADR(bRcvInCompl);
	p_bRcvNotStart ACCESS ADR(bRcvNotStart);
	p_bBAWidthEn ACCESS ADR(bBAWidthEn);
	p_bBASltEn ACCESS ADR(bBASltEn);
	p_bBFWidthEn ACCESS ADR(bBFWidthEn);
	p_bBFSltEn ACCESS ADR(bBFSltEn);
	p_sMcId ACCESS ADR(sMcId);
	p_sInterfaceId ACCESS ADR(sInterfaceId);
	p_sVersion ACCESS ADR(sVersion);
	p_eFailedBoard ACCESS ADR(eFailedBoard);
	p_sRecipeNm ACCESS ADR(sRecipeNm);
	p_diWidthInUM ACCESS ADR(diWidthInUM);
	p_diMinSltValue ACCESS ADR(diMinSltValue);
	p_diMaxSltValue ACCESS ADR(diMaxSltValue);
	p_diPitch ACCESS ADR(diPitch);
	p_diTtlSlt ACCESS ADR(diTtlSlt);
	p_diSltToSltInUM ACCESS ADR(diSltToSltInUM);
	p_udiSndBffrSize ACCESS ADR(udiSndBffrSize);
	p_udiRcvBffrSize ACCESS ADR(udiRcvBffrSize);
	p_udiAliveIdleTimeInSec ACCESS ADR(udiAliveIdleTimeInSec);
	p_tConnTimeOut ACCESS ADR(tConnTimeOut);
	p_diTransferInTO ACCESS ADR(diTransferInTO);
	p_bOpsRun ACCESS ADR(bOpsRun);
	p_bInterruptSen ACCESS ADR(bInterruptSen);
	p_udiFileKeepDay ACCESS ADR(udiFileKeepDay);
	p_sProgNm ACCESS ADR(sProgNm);
	p_bNtSettingsLoadDone ACCESS ADR(bNtSettingsLoadDone);
	p_bAccDataRdy ACCESS ADR(bAccDataRdy);
	p_sRmtMcId ACCESS ADR(sRmtMcId);
	p_bRmtPrep ACCESS ADR(bRmtPrep);
	p_bRmtEn ACCESS ADR(bRmtEn);
	p_bAccNewRcpCond ACCESS ADR(bAccNewRcpCond);
	p_sInfoMsg ACCESS ADR(sInfoMsg);
	p_sInfoMsg1 ACCESS ADR(sInfoMsg1);
	p_sInfoMsg2 ACCESS ADR(sInfoMsg2);
	p_bInternalUse ACCESS ADR(bInternalUse);
	p_sInternalRcv ACCESS ADR(sInternalRcv);
	pa_tyProdRcpList ACCESS ADR(a_tyProdRcpList);
	p_tyProdRcpCurrRcp ACCESS ADR(tyProdRcpCurrRcp);
	p_bMcParamMnlAccData ACCESS ADR(bMcParamMnlAccData);
	p_bUIAccData ACCESS ADR(bUIAccData);

	p_tyDSHermesCurrBASnd ACCESS ADR(tyBoardAvailableDummy);

	p_bManualRmvRoute ACCESS ADR(bManualRmvRoute);
	p_bReturnRoute ACCESS ADR(bReturnRoute);
	p_bNomRouteEn ACCESS ADR(bNomRouteEn);
	p_bProcessRouteEn ACCESS ADR(bProcessRouteEn);

	p_bReverseReceiveRoute ACCESS ADR(bReverseReceiveRoute);
	p_bReceiveReverseUSMcRdy ACCESS ADR(bReceiveReverseUSMcRdy);

	p_sTopBarcode  ACCESS ADR(sUITopBarcode);
	p_sBottomBarcode ACCESS ADR(sUIBottomBarcode);

	p_bHermesSwitchtoRvrseTransport ACCESS ADR(bSwitchtoReverseRcv);
END_ACTION
```

#### Act_Link.st
```iecst
(** 2019-06-04 **)
ACTION Act_Link:

	//Receive Alive Time
	p_tyParam.tRcvAlive	:= p_tyParam.tSndAlive * 2;

	//Transfer Complete
	IF (p_eLinkConvDir = ConvDirLToR) OR (p_eLinkConvDir = ConvDirLToL) THEN
		p_bRcvCompl	:= EDGENEG(p_bLinkDIRightSen);
	ELSE
		p_bRcvCompl	:= EDGENEG(p_bLinkDILeftSen);
	END_IF

	//Ready Receive
	p_bRdyRcv ACCESS p_OpsInvertStepUSCommTmr;

	//Ready Transport
	p_bRdyTransport	:= TRUE;

	//Accept New Recipe Condition
	p_bAccNewRcpCond	:= p_bLinkOpsRun = TRUE;

	//Routing
	p_bProcessRouteEn := p_bManualRmvRoute OR p_bReturnRoute OR p_bNomRouteEn;

	//Temporary Enable Reverse Receive
	p_bReverseReceiveRoute := TRUE;
	p_bReturnRoute := TRUE;
END_ACTION
```

#### Act_LinkAction.st
```iecst
(** 2019-04-09 **)
ACTION Act_LinkAction:

	IF p_bLinkStartupRun = TRUE THEN
		p_eAct ACCESS p_StartupUSHermesAct;
	ELSE
		p_eAct ACCESS ADR(eAct);

		IF EDGEPOS(p_eLinkMcParamUSCommMod = McSetCommModHermes) THEN
			bHermesRun	:= TRUE;
			bHermesStop	:= FALSE;
		END_IF

		IF EDGENEG(p_eLinkMcParamUSCommMod = McSetCommModHermes) THEN
			bHermesRun	:= FALSE;
			bHermesStop	:= TRUE;
		END_IF

		IF bHermesRun = TRUE THEN
			p_eAct	:= HermesActBGStartRun;

			IF (eStat = HermesActBGStartRun) AND (eStatus = Done) THEN
				p_eAct		:= HermesActIdle;
				bHermesRun	:= FALSE;
			END_IF
		END_IF

		IF bHermesStop = TRUE THEN
			p_eAct	:= HermesActBGStopRun;

			IF (eStat = HermesActBGStopRun) AND (eStatus = Done) THEN
				p_eAct		:= HermesActIdle;
				bHermesStop	:= FALSE;
			END_IF
		END_IF

	END_IF

	//Delete Old Log Files for 24 hours After Machine is Continuous Running 30 Days.

	fbDlyTmr(IN := TRUE);
	IF fbDlyTmr.Q THEN
		fbDeleteLogTmr (IN := TRUE);
		IF fbDeleteLogTmr.Q AND eStatus <> Busy THEN
			p_eAct := HermesActDeleteOldLog;
			IF eStat = HermesActDeleteOldLog AND eStatus = Done THEN
				p_eAct := HermesActIdle;
				fbDlyTmr (IN := FALSE);
				fbDeleteLogTmr (IN := FALSE);
			END_IF
		END_IF
	END_IF

END_ACTION
```

#### Act_Main_Disable.st
```iecst
(** 2019-03-15 **)
ACTION Act_Main_Disable:

	bConnected		:= FALSE;
	bHandshakeDone	:= FALSE;
	bAccDataReq		:= FALSE;
	bOverWriteSlt	:= FALSE;
	bOverWriteWidth	:= FALSE;
	bUSRdy			:= FALSE;
	bDSRdy			:= FALSE;
	bTransporting	:= FALSE;
	bStopTransport	:= FALSE;

END_ACTION
```

#### Cyclic.st
```iecst
(** 2020-09-10 **)
PROGRAM _CYCLIC

	IF bInitDone = FALSE THEN
		bInitDone	:= TRUE;

		Act_InitLocal;
		Act_InitGlobal;

	ELSIF bInitialDone = FALSE THEN
		IF p_bNtSettingsLoadDone = TRUE THEN
			bInitialDone	:= TRUE;

			Act_Initial;
		END_IF

	ELSE

		Act_RstErr;
		Act_LinkAction;
		Act_Action;
		Act_LinkEn;

		IF (p_bPrep = TRUE) AND (p_bEn = TRUE) AND (p_bDis = FALSE) THEN
			Act_Link;
			Act_Main;
			Act_Background;
		ELSE
			Act_Main_Disable;

			IF eStat <> HermesActIdle THEN
				eStatus	:= Done;
			ELSE
				eStatus	:= Idle;
			END_IF
		END_IF

		Act_CombineErr;
		Act_Alarm;
		Act_Alarm1;
		Act_Alarm2;
		Act_Alarm3;
		Act_Alarm4;
		Act_Alarm5;

	END_IF

END_PROGRAM
```

#### Init.st
```iecst
(** 2020-09-10 **)
PROGRAM _INIT

	(* Always Change If Project Change *)

	//Pass Address To Global Address For External Use
	//Action, State & Status
	p_USHermes2Stat		:= ADR(eStat);
	p_USHermes2Status	:= ADR(eMainStatus);
	p_USHermes2StatTxt	:= ADR(sStatTxt);

	//Alarm
	p_USHermes2AlmData	:= ADR(tyAlmData);
	p_USHermes2AlmData1	:= ADR(tyAlmData1);
	p_USHermes2AlmData2	:= ADR(tyAlmData2);
	p_USHermes2AlmData3	:= ADR(tyAlmData3);
	p_USHermes2AlmData4	:= ADR(tyAlmData4);
	p_USHermes2AlmData5	:= ADR(tyAlmData5);
	p_USHermes2InfoData	:= ADR(tyInfoData);

	//Output
	p_USHermes2TableDataBrdAvl			:= ADR(a_tyXMLTableDataBrdAvl);
	p_USHermes2TableDataBrdAvlTtlIdx	:= ADR(iXMLTableDataBrdAvlTtlIdx);
	p_USHermes2Connected				:= ADR(bConnected);
	p_USHermes2HandshakeDone			:= ADR(bHandshakeDone);
	p_USHermes2AccDataReq				:= ADR(bAccDataReq);
	p_USHermes2OverWriteSlt				:= ADR(bOverWriteSlt);
	p_USHermes2OverWriteWidth			:= ADR(bOverWriteWidth);
	p_USHermes2ReqRecipeNm				:= ADR(sReqRecipeNm);
	p_USHermes2ReqWidthInUM				:= ADR(diReqWidthInUM);
	p_USHermes2ReqMinSltValue			:= ADR(diReqMinSltValue);
	p_USHermes2ReqMaxSltValue			:= ADR(diReqMaxSltValue);
	p_USHermes2ReqPitch					:= ADR(diReqPitch);
	p_USHermes2USRdy					:= ADR(bUSRdy);
	p_USHermes2DSRdy					:= ADR(bDSRdy);
	p_USHermes2USGdRdy					:= ADR(bUSGdRdy);
	p_USHermes2DSGdRdy					:= ADR(bDSGdRdy);
	p_USHermes2Transporting				:= ADR(bTransporting);
	p_USHermes2StopTransport			:= ADR(bStopTransport);
	p_USHermes2BlkUS					:= ADR(bBlkUS);
	p_USHermes2InternalSnd				:= ADR(sInternalSnd);
	p_USHermes2AccDataMnl				:= ADR(bAccDataMnl);
	p_USHermes2StopTransportSnd 			:= ADR(bStopTransportSnd);

	p_USHermes2tyBoardAvailable			:= ADR(tyBoardAvailableRcv);
	p_USHermes2RcvBoardInfoOk        := ADR(bRcvBoardInfoOk);
	p_USHermes2RcvbBoardInfoIncompl  := ADR(bRcvBoardInfoIncompl);
	p_USHermes2BoardInfoData         := ADR(tySendBoardInfoAcc); //Pass "SendBoardInfo" data for DSHermes "BoardAvailable", for inserted PCB
	p_USHermes2BoardArrivedData		:= ADR(tyBoardArrivedInfo); //"BoardArrived" data for SupervisoryHermes

	//command
	p_USHermes2CommandParam				:= ADR(tyCommandParam);

	//Calling  on Reverse DS
	p_USHermes2ReverseDSSendBFId		:= ADR(bReverseDSSndBfWBrdID);
	p_USHermes2ProcessRouteTrigger		:= ADR(bTriggerUpdateRoute);

	//Block US Hermes
	p_USHermes2SwitchtoReverseRcv := ADR(bSwitchtoReverseReceive);
	(* Always Change If Project Change *)
	p_USHermes2BrdForecast			:= ADR(tyBoardForecastRcv);
	p_USHermes2BrdForecastRcv 		:= ADR(bBrdForecastRcv);
	p_USHermes2StopTransportSent    := ADR(bStopTransportSent);
	p_USHermes2StopTransportSentMsg	:= ADR(tyStopTransport);
	p_USHermes2BoardAvailableRcved   :=ADR(bBoardAvailableRcved);
END_PROGRAM
```

### DSHermes.var - Change By Project
```iecst
(*2020-09-10*)
(**)
(*Action & State & Status*)
VAR
	p_DSHermesStat : UDINT;
	p_DSHermesStatus : UDINT;
	p_DSHermesStatTxt : UDINT;
END_VAR
(**)
(*Alarm*)
VAR
	p_DSHermesAlmData : UDINT;
	p_DSHermesAlmData1 : UDINT;
	p_DSHermesAlmData2 : UDINT;
	p_DSHermesAlmData3 : UDINT;
	p_DSHermesAlmData4 : UDINT;
	p_DSHermesInfoData : UDINT;
END_VAR
(**)
(*Output*)
VAR
	p_DSHermesConnected : UDINT;
	p_DSHermesHandshakeDone : UDINT;
	p_DSHermesUSRdy : UDINT;
	p_DSHermesDSRdy : UDINT;
	p_DSHermesUSGdRdy : UDINT;
	p_DSHermesDSGdRdy : UDINT;
	p_DSHermesTransporting : UDINT;
	p_DSHermesStopTransport : UDINT;
	p_DSHermesInternalSnd : UDINT;
	p_DSHermesCommandParam : UDINT;
	p_DSHermesBrdAvlSnd : UDINT;
	p_DSHermesTransportFinish : UDINT;
	p_DSHermesTransportFinishMsg : UDINT;
END_VAR
```

### Program Logical/Hermes/DSHermes (IEC, version 1.00.0) - 1.00.0 - NtHermes v5.00.0 , NtTCP v5.00.0 , NtMessage v5.00.0

#### Init.st - Change By Project
```iecst
(** 2020-09-10 **)
PROGRAM _INIT

	(* Always Change If Project Change *)

	//Pass Address To Global Address For External Use
	//Action, State & Status
	p_DSHermesStat		:= ADR(eStat);
	p_DSHermesStatus	:= ADR(eMainStatus);
	p_DSHermesStatTxt	:= ADR(sStatTxt);

	//Alarm
	p_DSHermesAlmData	:= ADR(tyAlmData);
	p_DSHermesAlmData1	:= ADR(tyAlmData1);
	p_DSHermesAlmData2	:= ADR(tyAlmData2);
	p_DSHermesAlmData3	:= ADR(tyAlmData3);
	p_DSHermesAlmData4	:= ADR(tyAlmData4);
	p_DSHermesInfoData	:= ADR(tyInfoData);//detail mismatch machine ready and boardforecast

	//Output
	p_DSHermesConnected			:= ADR(bConnected);
	p_DSHermesHandshakeDone		:= ADR(bHandshakeDone);
	p_DSHermesUSRdy				:= ADR(bUSRdy);
	p_DSHermesDSRdy				:= ADR(bDSRdy);
	p_DSHermesUSGdRdy			:= ADR(bUSGdRdy);
	p_DSHermesDSGdRdy			:= ADR(bDSGdRdy);
	p_DSHermesTransporting		:= ADR(bTransporting);
	p_DSHermesStopTransport		:= ADR(bStopTransport);
	p_DSHermesInternalSnd		:= ADR(sInternalSnd);

	p_DSHermesTransportFinish	:=ADR(bTransportFinishedSnd);
	p_DSHermesTransportFinishMsg 	:=ADR(tyTransportFinished);
	//command
	p_DSHermesCommandParam			:= ADR(tyCommandParam);
	//route
	p_DSHermesBrdAvlSnd				:= ADR(tyBoardAvailableSnd);
	//p_DSHermesRcvReverseUSMcRdy		:= ADR(bDSHermesRcvReverseUSMcRdy);
	(* Always Change If Project Change *)

END_PROGRAM
```

#### Act_InitGlobal.st - Change By Project
```iecst
(** 2019-05-04 **)
ACTION Act_InitGlobal:

	(* Always Change If Project Change *)

	//Pass Data To Link
	p_bLinkStartupRun ACCESS p_StartupRun;
	p_eLinkMcParamDSCommMod ACCESS p_McParamDSCommMod;

	p_eLinkConvDir ACCESS p_NtParamProjConvDir;
	p_bLinkConvGdBrd ACCESS p_ConvGdBrd;
	p_bLinkDILeftSen ACCESS p_DIConvLftSen;
	p_bLinkDIRightSen ACCESS p_DIConvRgtSen;
	p_bLinkConvHvBrd ACCESS p_OpsInvertHvBrd;
	//Pass Data To Internal Use
	p_udiRstErr ACCESS p_RstErrReset;
	p_bPrep ACCESS p_NtParamHermesPrep;
	p_tyParam ACCESS p_HermesDSParam1;
	p_sIPAddr ACCESS p_HWInfoIPAddr;
	pa_usiMacAddr ACCESS p_HWInfoMacAddr;
	p_tyDTStructure ACCESS p_TimeCurrDTStruct;
	p_dtCurrDT ACCESS p_TimeCurrDT;
	p_sMcId ACCESS p_McParamMcNm;
	p_sRecipeNm ACCESS p_ProdRcpCurrRcp0Nm;
	p_sRecipeZone1Nm ACCESS p_ProdRcpCurrRcp1Nm;
	//p_sWorkOrderId ACCESS p_SvyHermesWorkOrderId; //Work Order Id from SupervisoryHermes
	//p_sBatchId ACCESS p_SvyHermesBatchId; //Batch Id from SupervisoryHermes
	p_diWidthInUM ACCESS p_ProdRcpCurrRcp0Width;
	p_diWidthZone1InUM ACCESS p_ProdRcpCurrRcp1Width;
	p_udiAliveIdleTimeInSec ACCESS p_NtParamDSHermesAliveTmInSec;
	p_tConnTimeOut ACCESS p_NtParamDSHermesConnTO;
	p_diTransferInTO ACCESS p_McParamTranOutErrDlyTm;
	pa_tyXMLTableDataBrdAvl ACCESS p_HermesBrdAvlDataTableLastZ;
	p_iXMLTableDataBrdAvlTtlIdx ACCESS p_HermesBrdAvlDataTtlIdxLastZ;
	p_bNewBrdAvlFirstZone ACCESS p_HermesBrdAvlDataNewBrdAvl1stZ;
	p_bNewBrdAvlLastZone ACCESS p_HermesBrdAvlDataNewBrdAvlLastZ;
	p_bOpsRun ACCESS p_OpsRun;
	p_bInterruptSen ACCESS p_DIConvRgtSen;
	p_udiFileKeepDay ACCESS p_NtParamDSHermesFileKeepDay;
	p_sRetainFileName ACCESS p_NtParamDSHermesRetainFileNm;
	p_sProgNm ACCESS p_NtParamDSHermesProgNm;
	p_bNtSettingsLoadDone ACCESS p_StartupNtSettingsLoadDone;
	p_sRmtMcId ACCESS p_RmtHermesCurrentConfMcId;
	p_bRmtPrep ACCESS p_NtParamHermesRmtPrep;
	p_bRmtEn ACCESS p_McParamHermesRmtEn;

	p_bUSHermesStopTransport ACCESS p_USHermesStopTransportSnd;

	p_tyUSHermestyBoardAvailable ACCESS p_USHermestyBoardAvailable;
	p_bNtParamProjInvertOncePrep ACCESS p_NtParamProjInvertOncePrep;
	p_bNtParamProjInvertTwicePrep ACCESS p_NtParamProjInvertTwicePrep;

	//for reverse condition
	//p_bUSHermesReverseDSSendBFId ACCESS p_USHermesReverseDSSendBFId;
	//p_bUSHermesProcessRouteTrigger ACCESS p_USHermesProcessRouteTrigger;
	p_usiUSHermesReverseDSSendBFId ACCESS p_HermesReverseDS1SendBFId;//p_USHermes2ReverseDSSendBFId;
	p_bUSHermesProcessRouteTrigger ACCESS p_USHermes2ProcessRouteTrigger;
	p_tySvyHermesSendWorkOrderInfo ACCESS p_SvyHermesSendWorkOrderInfo; //SvyRcvBoardInfo from Supervisor, used to generate B.A for inserted PCB
	pa_RevtyXMLTableDataBrdAvl  ACCESS p_USHermesTableDataBrdAvl;
	p_ReviXMLTableDataBrdAvlTtlIdx ACCESS  p_USHermesTableDataBrdAvlTtlIdx;

	//BoardForecast
	p_tyUSBoardArrivedData  ACCESS p_USHermesBoardArrivedData;
	//Board Available

	p_bRcvBoardInfo ACCESS p_USHermesRcvBoardInfoOk;
	p_tyBoardInfoData ACCESS p_USHermesBoardInfoData;

	p_bConvInitDone ACCESS p_OpsInvertStepInitConv;

	p_bHermesSwitchtoRvrseTransport ACCESS p_HermesSwitchtoReverseTransport;
	(* Always Change If Project Change *)

END_ACTION
```

#### InputRef_Link.var - Change By Project
```iecst
(*2019-04-09*)
(**)
VAR
	p_bLinkStartupRun : REFERENCE TO BOOL;
	p_eLinkMcParamDSCommMod : REFERENCE TO eMcSetCommMod;
	bHermesRun : BOOL;
	bHermesStop : BOOL;
END_VAR
(**)
VAR
	p_eLinkConvDir : REFERENCE TO eConvDir;
	p_bLinkConvGdBrd : REFERENCE TO BOOL;
	p_bLinkDILeftSen : REFERENCE TO BOOL;
	p_bLinkDIRightSen : REFERENCE TO BOOL;
	p_bLinkConvHvBrd : REFERENCE TO BOOL;
END_VAR
(**)
VAR
	fbDlyTmr : TON := (PT:=T#5s);
	fbDeleteLogTmr : TON := (PT:=T#24h);
END_VAR
```

#### Act_LinkAction.st - Change By Project
```iecst
(** 2021-08-01 **)
ACTION Act_LinkAction:

	IF p_bLinkStartupRun = TRUE THEN
		p_eAct ACCESS p_StartupDSHermesAct;
	ELSE
		p_eAct ACCESS ADR(eAct);

		IF EDGEPOS(p_eLinkMcParamDSCommMod = McSetCommModHermes) THEN
			bHermesRun	:= TRUE;
			bHermesStop	:= FALSE;
		END_IF

		IF EDGENEG(p_eLinkMcParamDSCommMod = McSetCommModHermes) THEN
			bHermesRun	:= FALSE;
			bHermesStop	:= TRUE;
		END_IF

		IF bHermesRun = TRUE THEN
			p_eAct	:= HermesActBGStartRun;

			IF (eStat = HermesActBGStartRun) AND (eStatus = Done) THEN
				p_eAct		:= HermesActIdle;
				bHermesRun	:= FALSE;
			END_IF
		END_IF

		IF bHermesStop = TRUE THEN
			p_eAct	:= HermesActBGStopRun;

			IF (eStat = HermesActBGStopRun) AND (eStatus = Done) THEN
				p_eAct		:= HermesActIdle;
				bHermesStop	:= FALSE;
			END_IF
		END_IF

	END_IF

	//Delete Old Hermese Log Files for 24 hours After Machine is Continuous Running 7 Days.
	fbDlyTmr(IN := TRUE);
	IF fbDlyTmr.Q THEN
		fbDeleteLogTmr (IN := TRUE);
		IF fbDeleteLogTmr.Q AND eStatus <> Busy THEN
			p_eAct := HermesActDeleteOldLog;
			IF eStat = HermesActDeleteOldLog AND eStatus = Done THEN
				p_eAct := HermesActIdle;
				fbDlyTmr (IN := FALSE);
				fbDeleteLogTmr (IN := FALSE);
			END_IF
		END_IF
	END_IF

END_ACTION
```

#### Act_Link.st - Change By Project
```iecst
(** 2019-04-08 **)
ACTION Act_Link:

	//Receive Alive Time
	p_tyParam.tRcvAlive	:= p_tyParam.tSndAlive * 2;

	//Ready Send //need to uncomment back
	p_bRdySnd ACCESS p_OpsInvertStepDSCommTmr;

	//boardforecast
	bNewProduct := EDGEPOS(p_sRecipeNm <> p_sRecipeZone1Nm) AND p_bLinkStartupRun = FALSE;
	bNewWidth := EDGEPOS(p_diWidthInUM <> p_diWidthZone1InUM) AND p_bLinkStartupRun = FALSE;
	bAllZoneEmpty := p_bLinkDIRightSen = FALSE AND p_bLinkDILeftSen = FALSE AND p_bLinkConvHvBrd = FALSE;

	//Transfer Finished
	IF NOT(p_bHermesSwitchtoRvrseTransport) THEN //(p_eLinkConvDir = ConvDirLToR) OR (p_eLinkConvDir = ConvDirRToR) THEN
		IF EDGENEG(p_bLinkDIRightSen) THEN
			p_bSndCompl	:= TRUE;
		END_IF
		bFirstZoneHaveBoard :=  p_bLinkDILeftSen;
		bFirstZoneEndSen :=  p_bLinkDIRightSen ;
	ELSE
		IF EDGENEG(p_bLinkDILeftSen) THEN
			p_bSndCompl	:= TRUE;
		END_IF
		bFirstZoneHaveBoard := p_bLinkDIRightSen ;
		bFirstZoneEndSen :=  p_bLinkDILeftSen ;
	END_IF

	//Good Bad Board
	IF p_bLinkConvGdBrd = TRUE THEN
		p_eFailedBoard	:= HermesGoodBoard;
	ELSE
		p_eFailedBoard	:= HermesFailedBoard;
	END_IF

	//Flip Board
//	IF p_tyUSHermestyBoardAvailable.tyData.eFlippedBoard = 2 THEN
//		p_eFlippedBoard := 1;
//
//	ELSIF p_tyUSHermestyBoardAvailable.tyData.eFlippedBoard = 1 THEN
//		p_eFlippedBoard := 2;
//
//	ELSE
//		p_eFlippedBoard := 0;
//	END_IF

	//first zone have board
	//Machine First Zone have board
	//p_bFirstZoneHaveBoard := (p_bUSHermesStopTransport AND p_bOpsGConvHvBrd) OR (p_bOpsGConvHvBrd AND p_bUSHermesTransporting = FALSE); //Zone 1 have board, either PCB_In from upstream Or Manually load PCB at Zone 1

END_ACTION
```

#### Cyclic.st - Do Not Change!!!
```iecst
(** 2020-09-10 **)
PROGRAM _CYCLIC

	IF bInitDone = FALSE THEN
		bInitDone	:= TRUE;

		Act_InitLocal;
		Act_InitGlobal;

	ELSIF bInitialDone = FALSE THEN
		IF p_bNtSettingsLoadDone = TRUE THEN
			bInitialDone	:= TRUE;

			Act_Initial;
		END_IF

	ELSE

		Act_RstErr;
		Act_LinkAction;
		Act_Action;
		Act_LinkEn;

		IF (p_bPrep = TRUE) AND (p_bEn = TRUE) AND (p_bDis = FALSE) THEN
			Act_Link;
			Act_Main;
			Act_Background;
			Act_Background_ProcessData;
		ELSE
			Act_Main_Disable;

			IF eStat <> HermesActIdle THEN
				eStatus	:= Done;
			ELSE
				eStatus	:= Idle;
			END_IF
		END_IF

		Act_CombineErr;
		Act_Alarm;
		Act_Alarm1;
		Act_Alarm2;
		Act_Alarm3;
		Act_Alarm4;

	END_IF

END_PROGRAM
```

#### Act_InitLocal.st - Do Not Change!!!
```iecst
(** 2019-06-10 **)
ACTION Act_InitLocal:

	//Input Reference Link To Local Variable
	p_eAct ACCESS ADR(eAct);
	p_udiRstErr ACCESS ADR(udiRstErr);
	p_bPrep ACCESS ADR(bPrep);
	p_bEn ACCESS ADR(bEn);
	p_bDis ACCESS ADR(bDis);
	p_tyParam ACCESS ADR(tyParam);
	p_sIPAddr ACCESS ADR(sIPAddr);
	pa_usiMacAddr ACCESS ADR(a_usiMacAddr);
	p_tyDTStructure ACCESS ADR(tyDTStructure);
	p_dtCurrDT ACCESS ADR(dtCurrDT);
	p_bRdySnd ACCESS ADR(bRdySnd);
	p_bSndCompl ACCESS ADR(bSndCompl);
	p_bSndIncompl ACCESS ADR(bSndInCompl);
	p_bSndNotStart ACCESS ADR(bSndNotStart);
	p_bBAWidthEn ACCESS ADR(bBAWidthEn);
	p_bBASltEn ACCESS ADR(bBASltEn);
	p_bBFWidthEn ACCESS ADR(bBFWidthEn);
	p_bBFSltEn ACCESS ADR(bBFSltEn);
	p_sMcId ACCESS ADR(sMcId);
	p_sInterfaceId ACCESS ADR(sInterfaceId);
	p_sVersion ACCESS ADR(sVersion);
	p_eFailedBoard ACCESS ADR(eFailedBoard);
	p_sRecipeNm ACCESS ADR(sRecipeNm);
	p_eFlippedBoard ACCESS ADR(eFlippedBoard);
	p_sTopBarcode ACCESS ADR(sTopBarcode);
	p_sBottomBarcode ACCESS ADR(sBottomBarcode);
	p_rLength ACCESS ADR(rLength);
	p_rThickness ACCESS ADR(rThickness);
	p_rConveyorSpeed ACCESS ADR(rConveyorSpeed);
	p_rTopClearanceHeight ACCESS ADR(rTopClearanceHeight);
	p_rBottomClearanceHeight ACCESS ADR(rBottomClearanceHeight);
	p_rWeight ACCESS ADR(rWeight);
	p_sWorkOrderId ACCESS ADR(sWorkOrderId);
	p_sBatchId ACCESS ADR(sBatchId);
	p_diWidthInUM ACCESS ADR(diWidthInUM);
	p_diMinSltValue ACCESS ADR(diMinSltValue);
	p_diMaxSltValue ACCESS ADR(diMaxSltValue);
	p_diPitch ACCESS ADR(diPitch);
	p_diTtlSlt ACCESS ADR(diTtlSlt);
	p_diSltToSltInUM ACCESS ADR(diSltToSltInUM);
	p_udiSndBffrSize ACCESS ADR(udiSndBffrSize);
	p_udiRcvBffrSize ACCESS ADR(udiRcvBffrSize);
	p_udiAliveIdleTimeInSec ACCESS ADR(udiAliveIdleTimeInSec);
	p_tConnTimeOut ACCESS ADR(tConnTimeOut);
	p_diTransferInTO ACCESS ADR(diTransferInTO);
	pa_tyXMLTableDataBrdAvl ACCESS ADR(a_tyXMLTableDataBrdAvl);
	p_iXMLTableDataBrdAvlTtlIdx ACCESS ADR(iXMLTableDataBrdAvlTtlIdx);
	p_bNewBrdAvlFirstZone ACCESS ADR(bNewBrdAvl);
	p_bOpsRun ACCESS ADR(bOpsRun);
	p_bInterruptSen ACCESS ADR(bInterruptSen);
	p_udiFileKeepDay ACCESS ADR(udiFileKeepDay);
	p_sProgNm ACCESS ADR(sProgNm);
	p_bNtSettingsLoadDone ACCESS ADR(bNtSettingsLoadDone);
	p_sRmtMcId ACCESS ADR(sRmtMcId);
	p_bRmtPrep ACCESS ADR(bRmtPrep);
	p_bRmtEn ACCESS ADR(bRmtEn);
	p_bInternalUse ACCESS ADR(bInternalUse);
	p_sInternalRcv ACCESS ADR(sInternalRcv);
	p_eFlippedBoard ACCESS ADR(eFlippedBoard);
	p_tyUSHermestyBoardAvailable ACCESS ADR(tyUSHermestyBoardAvailable);
	p_bManualInsertData ACCESS ADR (bDummy);
	//p_bManualInsertData  ACCESS p_ManualInsertData;
	p_rMcCycleTm ACCESS ADR(rMachineCycleTime);
	p_rAWCycleTm ACCESS ADR(rAWCycleTm);
	//Route
	p_bProcessRouteEn ACCESS ADR(bProcessRouteEn);
	p_bManualRmvRoute ACCESS ADR(bManualRmvRoute);
	p_bReturnRoute ACCESS ADR(bReturnRoute);
	p_bNomRouteEn ACCESS ADR(bNomRouteEn);

	p_bReverseSentRoute ACCESS ADR(bReverseSentRoute);
	p_usiUSHermesReverseDSSendBFId ACCESS ADR(usiUSHermesReverseDSSendBFId);
	p_bUSHermesProcessRouteTrigger ACCESS ADR(bUSHermesProcessRouteTrigger);

END_ACTION
```

#### Act_Background.st - Do Not Change!!!
```iecst
(** 2021-08-01 **)
ACTION Act_Background:

	IF bRun = TRUE THEN
		IF udiSvrIdent = 0 THEN
			IF p_bInternalUse = FALSE THEN
				Act_Background_TCPCreateSvr;

				tyParamOld	:= p_tyParam;
			ELSE
				udiSvrIdent	:= 1;
			END_IF

		ELSE
			IF bRstConnection = FALSE THEN

				Act_Background_ChgConfig;

				IF udiClntIdent = 0 THEN
					IF p_bInternalUse = FALSE THEN
						Act_Background_TCPListen;
					ELSE
						udiClntIdent	:= 1;
					END_IF

				ELSE
					Act_Background_TCPRcv;

					Act_Background_NotificationRcv;

					Act_Background_IllegalMsg;
					Act_Background_ChkParamRcv;
					Act_Background_CmpParamRcv;

					IF bHandshakeDone = TRUE THEN
						IF (p_tyParam.tSndAlive <> T#0s) AND (p_tyParam.tRcvAlive <> T#0s) THEN
							IF tyServiceDescriptionRcv.tyData.tySupportedFeatures.bFeatureCheckAliveResponse = TRUE AND p_tyParam.bFeatureCheckAliveResponse = TRUE THEN
								Act_Background_ChkAliveSendPing;
								Act_Background_ChkAliveRcvPing;
							ELSE
								Act_Background_ChkAlive;
							END_IF
						ELSE
							fbCheckAlive(bEn := FALSE);
							fbCheckAliveSendPing(bEn := FALSE);
							fbCheckAliveRcvPing(bEn := FALSE);
						END_IF
					END_IF

					Act_Background_BoardForecast;
					Act_Background_SendBoardInfo;
					//Act_Background_Route;

					Act_Background_Sequence;
					Act_Background_SequenceTO;
					Act_Background_Err;

					Act_Background_Command;

					Act_Background_TCPSend;

					Act_Background_Log;

				END_IF

			ELSE
				IF udiClntIdent <> 0 THEN
					Act_Background_TCPCloseClnt;
				ELSE
					IF udiSvrIdent <> 0 THEN
						Act_Background_TCPCloseSvr;
					END_IF
				END_IF

			END_IF

			//Second Client Connected
			IF udiClntIdentExtra = 0 THEN

			ELSE

			END_IF

		END_IF

		Act_Background_Stop;

	END_IF

	IF EDGENEG(bRun) OR EDGENEG(udiSvrIdent = 0) THEN
		//Reset
		fbCreateSvr(bEn := FALSE);
	END_IF

	IF EDGENEG(bRun) OR EDGENEG(udiClntIdent = 0) THEN
		//Reset
		fbListen(bEn := FALSE);

		bConnected	:= bRun;
	END_IF

	IF EDGENEG(bRun) OR EDGENEG(udiSvrIdent <> 0) OR EDGENEG(udiClntIdent <> 0) THEN
		fbRcv(bEn := FALSE);
		fbSequenceDS(bEn := FALSE);
		fbSequenceTO(bEn := FALSE);
		fbCheckAlive(bEn := FALSE);
		fbCheckAliveSendPing(bEn := FALSE);
		fbCheckAliveRcvPing(bEn := FALSE);
		fbSend(bEn := FALSE);

		fbFileAppend1(bEn := FALSE);
		iWriteLogStep	:= 0;

		bConnected		:= FALSE;
		bHandshakeDone	:= FALSE;
		bRstState		:= FALSE;
		bUSRdy			:= FALSE;
		bDSRdy			:= FALSE;
		bTransporting	:= FALSE;
		bStopTransport	:= FALSE;

		memset(ADR(tyMsgTypeRcv) , 0 , SIZEOF(tyMsgTypeRcv));
		memset(ADR(a_eMsgSend) , 0 , SIZEOF(a_eMsgSend));
		udiMsgSendBffr	:= 0;
	END_IF

	IF EDGENEG(bRun) OR EDGENEG(udiSvrIdent <> 0) THEN
		bRstConnection	:= FALSE;
		fbCloseSvr(bEn := FALSE);
	END_IF

	IF EDGENEG(bRun) OR EDGENEG(udiClntIdent <> 0) THEN
		fbCloseClnt(bEn := FALSE);
	END_IF

	//Reset Error
	IF (eStatus1 = Error) AND bRstErr THEN
		eStatus1	:= Idle;
		udiStatus1	:= 0;

		fbCreateSvr(bEn := FALSE);
		fbListen(bEn := FALSE);
		fbRcv(bEn := FALSE);
		fbSequenceDS(bEn := FALSE);
		fbSend(bEn := FALSE);
		fbCloseSvr(bEn := FALSE);
		fbCloseClnt(bEn := FALSE);
		fbCheckAlive(bEn := FALSE);
		fbCheckAliveSendPing(bEn := FALSE);
		fbCheckAliveRcvPing(bEn := FALSE);
		fbSequenceTO(bEn := FALSE);

		fbFileAppend1(bEn := FALSE);
		iWriteLogStep	:= 0;

		bConnected		:= FALSE;
		bHandshakeDone	:= FALSE;
		bRstConnection	:= FALSE;
		bRstState		:= FALSE;
		bUSRdy			:= FALSE;
		bDSRdy			:= FALSE;
		bTransporting	:= FALSE;
		bStopTransport	:= FALSE;

		memset(ADR(tyMsgTypeRcv) , 0 , SIZEOF(tyMsgTypeRcv));
		memset(ADR(a_eMsgSend) , 0 , SIZEOF(a_eMsgSend));
		udiMsgSendBffr	:= 0;
	END_IF

	IF (eStatus2 = Error) AND bRstErr THEN
		eStatus2	:= Idle;
		udiStatus2	:= 0;

		fbSequenceTO(bEn := FALSE);

	END_IF

	IF (eStatus3 = Error) AND bRstErr THEN
		eStatus3	:= Idle;
		udiStatus3	:= 0;

		fbFileAppend1(bEn := FALSE);
		iWriteLogStep	:= 0;
	END_IF

END_ACTION
```

#### Act_Background_TCPCreateSvr.st - Do Not Change!!!
```iecst
(** 2021-08-01 **)
ACTION Act_Background_TCPCreateSvr:

	IF eStatus1 <> Error THEN

		//Create Server
		fbCreateSvr.sSvrIP				:= p_sIPAddr;
		fbCreateSvr.uiSvrPort			:= p_tyParam.uiSvrPort;
		fbCreateSvr(bEn := TRUE);

		IF fbCreateSvr.udiStatus = 0 THEN
			udiSvrIdent	:= fbCreateSvr.udiTCPIdent;
			fbCreateSvr(bEn := FALSE);

		ELSIF fbCreateSvr.udiStatus < 65534 THEN
			eStatus1	:= Error;

			IF fbCreateSvr.udiStatus = 2300 THEN
				udiStatus1	:= 10000;	//Invalid Ident While Creating Server
			ELSIF fbCreateSvr.udiStatus = 2302 THEN
				udiStatus1	:= 10001;	//Setting Keep Alive Interval Time Error While Creating Server
			ELSIF fbCreateSvr.udiStatus = 2303 THEN
				udiStatus1	:= 10002;	//Setting Keep Alive Idle Time Error While Creating Server
			ELSIF fbCreateSvr.udiStatus = 2304 THEN
				udiStatus1	:= 10003;	//Setting Keep Alive Count Error While Creating Server
			ELSIF fbCreateSvr.udiStatus = 2305 THEN
				udiStatus1	:= 10004;	//Setting Keep Alive Error While Creating Server
			ELSIF fbCreateSvr.udiStatus = 2306 THEN
				udiStatus1	:= 10005;	//Setting Receive Buffer Error While Creating Server
			ELSIF fbCreateSvr.udiStatus = 2307 THEN
				udiStatus1	:= 10006;	//Setting Send Buffer Error While Creating Server
			ELSIF fbCreateSvr.udiStatus = 2308 THEN
				udiStatus1	:= 10007;	//Setting No Waiting Error While Creating Server
			ELSIF fbCreateSvr.udiStatus = 2309 THEN
				udiStatus1	:= 10008;	//TCP Open Port Error While Creating Server
			ELSIF fbCreateSvr.udiStatus = 2310 THEN
				udiStatus1	:= 10009;	//Closing TCP Error While Creating Server
			ELSE
				udiStatus1	:= fbCreateSvr.udiStatus;
			END_IF

		END_IF

	END_IF

END_ACTION
```

#### Act_Background_TCPListen.st - Do Not Change!!!
```iecst
(** 2021-08-01 **)
ACTION Act_Background_TCPListen:

	IF eStatus1 <> Error AND eStatus2 <> Error THEN

		fbListen.udiSvrIdent	:= udiSvrIdent;
		fbListen(bEn := TRUE);

		IF fbListen.udiStatus = 0 THEN
			udiClntIdent	:= fbListen.udiClntIdent;
			fbListen(bEn := FALSE);

		ELSIF fbListen.udiStatus = 2311 THEN //No Client Connected
			fbListen(bEn := FALSE);

		ELSIF fbListen.udiStatus = 2312 OR (bConnected=FALSE) THEN
			udiStatus4	:= 10012;	//DS Hermes Connection Lost
			fbListen(bEn := FALSE); //add

		ELSIF fbListen.udiStatus < 65534 THEN
			eStatus1	:= Error;

			IF fbListen.udiStatus = 2300 THEN
				udiStatus1	:= 10010;	//Invalid Ident While Listening Client
			ELSE
				udiStatus1	:= fbListen.udiStatus;
			END_IF

		END_IF

	END_IF

END_ACTION
```

#### Act_Background_TCPRcv.st - Do Not Change!!!
```iecst
(** 2021-08-01 **)
ACTION Act_Background_TCPRcv:

	IF eStatus1 <> Error THEN

		//Receive Data
		IF p_bInternalUse = FALSE THEN
			fbRcv.udiTCPIdent	:= udiClntIdent;
			fbRcv(bEn := TRUE);
		ELSE
			sRcv	:= p_sInternalRcv;
		END_IF

		IF (fbRcv.udiStatus = 0) OR ((p_bInternalUse = TRUE) AND (LEN(sRcv) > 0)) THEN

			fLogDTConvert(ADR(sDT) , p_dtCurrDT);
			memset(ADR(a_sLogList[udiLogCntr]) , 0 , SIZEOF(a_sLogList[udiLogCntr]));
			memcpy(ADR(a_sLogList[udiLogCntr]) + LEN(a_sLogList[udiLogCntr]) , ADR(sDT) , LEN(sDT));
			memcpy(ADR(a_sLogList[udiLogCntr]) + LEN(a_sLogList[udiLogCntr]) , ADR('$r$n') , LEN('$r$n'));
			memcpy(ADR(a_sLogList[udiLogCntr]) + LEN(a_sLogList[udiLogCntr]) , ADR('RCV_FRM_DS$r$n') , LEN('RCV_FRM_DS$r$n'));
			memcpy(ADR(a_sLogList[udiLogCntr]) + LEN(a_sLogList[udiLogCntr]) , ADR(sRcv) , LEN(sRcv));
			memcpy(ADR(a_sLogList[udiLogCntr]) + LEN(a_sLogList[udiLogCntr]) , ADR('$r$n$r$n') , LEN('$r$n$r$n'));

			udiLogCntr	:= udiLogCntr + 1;
			IF udiLogCntr = 11 THEN
				udiLogCntr	:= 1;
			END_IF

			fXMLConvertToTable(ADR(sRcv) , LEN(sRcv) , ADR(a_tyXMLTableDataRcv) , ADR(a_tyXMLTableDataRcv[0].sTitle) , SIZEOF(a_tyXMLTableDataRcv[0].sTitle) , ADR(a_tyXMLTableDataRcv[0].sValue) , SIZEOF(a_tyXMLTableDataRcv[0].sValue) , ADR(a_tyXMLTableDataRcv[0].uiSize) , SIZEOF(a_tyXMLTableDataRcv[0]) , SIZEOF(a_tyXMLTableDataRcv) / SIZEOF(a_tyXMLTableDataRcv[0]) , ADR(udiXMLTableWriteIdx));

			fbParseXMLTable.iTotalIdxWrite	:= UDINT_TO_INT(udiXMLTableWriteIdx);
			fbParseXMLTable;

			IF fbParseXMLTable.tyMsgType.bCheckAlive = TRUE THEN
				tyMsgTypeRcv.bCheckAlive	:= TRUE;
				tyCheckAliveRcv				:= fbParseXMLTable.tyCheckAlive;
			END_IF

			IF fbParseXMLTable.tyMsgType.bCheckAlivePing = TRUE THEN
				tyMsgTypeRcv.bCheckAlivePing	:= TRUE;
				tyCheckAlivePingRcv				:= fbParseXMLTable.tyCheckAlivePing;
			END_IF

			IF fbParseXMLTable.tyMsgType.bCheckAlivePong = TRUE THEN
				tyMsgTypeRcv.bCheckAlivePong	:= TRUE;
				tyCheckAlivePongRcv				:= fbParseXMLTable.tyCheckAlivePong;
			END_IF

			IF fbParseXMLTable.tyMsgType.bServiceDescription = TRUE THEN
				tyMsgTypeRcv.bServiceDescription	:= TRUE;
				tyServiceDescriptionRcv				:= fbParseXMLTable.tyServiceDescription;
			END_IF

			IF fbParseXMLTable.tyMsgType.bNotification = TRUE THEN
				tyMsgTypeRcv.bNotification	:= TRUE;
				tyNotificationRcv			:= fbParseXMLTable.tyNotification;
			END_IF

			IF fbParseXMLTable.tyMsgType.bBoardAvailable = TRUE THEN
				tyMsgTypeRcv.bBoardAvailable	:= TRUE;
				tyBoardAvailableRcv				:= fbParseXMLTable.tyBoardAvailable;

				memset(ADR(a_tyXMLTableDataBrdAvl) , 0 , SIZEOF(a_tyXMLTableDataBrdAvl));
				memcpy(ADR(a_tyXMLTableDataBrdAvl) , ADR(a_tyXMLTableDataRcv) + (fbParseXMLTable.iBoardAvailableFirstIdx * SIZEOF(a_tyXMLTableDataRcv[0])) , (fbParseXMLTable.iBoardAvailableLastIdx - fbParseXMLTable.iBoardAvailableFirstIdx + 1) * SIZEOF(a_tyXMLTableDataRcv[0]));

			END_IF

			IF fbParseXMLTable.tyMsgType.bRevokeBoardAvailable = TRUE THEN
				tyMsgTypeRcv.bRevokeBoardAvailable	:= TRUE;
			END_IF

			IF fbParseXMLTable.tyMsgType.bMachineReady = TRUE THEN
				tyMsgTypeRcv.bMachineReady	:= TRUE;
				tyMachineReady				:= fbParseXMLTable.tyMachineReady;
			END_IF

			IF fbParseXMLTable.tyMsgType.bRevokeMachineReady = TRUE THEN
				tyMsgTypeRcv.bRevokeMachineReady	:= TRUE;
			END_IF

			IF fbParseXMLTable.tyMsgType.bStartTransport = TRUE THEN
				tyMsgTypeRcv.bStartTransport	:= TRUE;
				tyStartTransport				:= fbParseXMLTable.tyStartTransport;
			END_IF

			IF fbParseXMLTable.tyMsgType.bStopTransport = TRUE THEN
				tyMsgTypeRcv.bStopTransport	:= TRUE;
				tyStopTransport				:= fbParseXMLTable.tyStopTransport;
			END_IF

			IF fbParseXMLTable.tyMsgType.bTransportFinished = TRUE THEN
				tyMsgTypeRcv.bTransportFinished	:= TRUE;
				tyTransportFinished				:= fbParseXMLTable.tyTransportFinished;
			END_IF

			IF fbParseXMLTable.tyMsgType.bSetConfiguration = TRUE THEN
				tyMsgTypeRcv.bSetConfiguration	:= TRUE;
				tySetConfiguration				:= fbParseXMLTable.tySetConfiguration;
			END_IF

			IF fbParseXMLTable.tyMsgType.bGetConfiguration = TRUE THEN
				tyMsgTypeRcv.bGetConfiguration	:= TRUE;
			END_IF

			IF fbParseXMLTable.tyMsgType.bCurrentConfiguration = TRUE THEN
				tyMsgTypeRcv.bCurrentConfiguration	:= TRUE;
				tyCurrentConfiguration				:= fbParseXMLTable.tyCurrentConfiguration;
			END_IF

			IF fbParseXMLTable.tyMsgType.bBoardForecast = TRUE THEN
				tyMsgTypeRcv.bBoardForecast	:= TRUE;
				tyBoardForecastRcv				:= fbParseXMLTable.tyBoardForecast;
			END_IF

			IF fbParseXMLTable.tyMsgType.bQueryBoardInfo = TRUE THEN
				tyMsgTypeRcv.bQueryBoardInfo	:= TRUE;
				tyQueryBoardInfo				:= fbParseXMLTable.tyQueryBoardInfo;
			END_IF

			IF fbParseXMLTable.tyMsgType.bSendBoardInfo = TRUE THEN
				tyMsgTypeRcv.bSendBoardInfo	:= TRUE;
				tySendBoardInfo				:= fbParseXMLTable.tySendBoardInfo;
			END_IF

			IF fbParseXMLTable.tyMsgType.bCommand = TRUE THEN
				tyMsgTypeRcv.bCommand	:= TRUE;
				tyCommandRcv				:= fbParseXMLTable.tyCommand;
			END_IF

			fbRcv(bEn := FALSE);

			memset(ADR(sRcv) , 0 , SIZEOF(sRcv));

		ELSIF (fbRcv.udiStatus = 2317) AND (p_bInternalUse = FALSE) THEN
			fbRcv(bEn := FALSE);

			memset(ADR(sRcv) , 0 , SIZEOF(sRcv));

		ELSIF (fbRcv.udiStatus = 2316) AND (p_bInternalUse = FALSE) THEN
			bRstConnection	:= TRUE;

			memset(ADR(sRcv) , 0 , SIZEOF(sRcv));

		ELSIF (fbRcv.udiStatus = 2318) AND (p_bInternalUse = FALSE) THEN
			bRstConnection	:= TRUE;

			memset(ADR(sRcv) , 0 , SIZEOF(sRcv));

		ELSIF (fbRcv.udiStatus < 65534) AND (p_bInternalUse = FALSE) THEN
			eStatus1	:= Error;

			IF fbRcv.udiStatus = 2300 THEN
				udiStatus1	:= 10014;	//Invalid Ident While Receiving Data
			ELSIF fbRcv.udiStatus = 2319 THEN
				udiStatus1	:= 10015;	//TCP Receive Data Error While Receiving Data
			ELSE
				udiStatus1	:= fbRcv.udiStatus;
			END_IF

			memset(ADR(sRcv) , 0 , SIZEOF(sRcv));

		END_IF

	END_IF

END_ACTION
```

#### Act_Background_ChkParamRcv.st - Do Not Change!!!
```iecst
(** 2019-03-25 **)
ACTION Act_Background_ChkParamRcv:

	IF eStatus2 <> Error THEN

		//Check Parameter Receive
		IF tyMsgTypeRcv.bServiceDescription = TRUE THEN
			udiStatus2	:= fHermesChkParamSD(tyServiceDescriptionRcv , p_tyParam.iLaneID);

			IF udiStatus2 = 2731 THEN
				udiStatus2	:= 0;
			END_IF

			IF udiStatus2 <> 0 THEN
				eStatus2	:= Error;

				IF udiStatus2 = 2726 THEN
					udiStatus2	:= 10086;	//LaneId Mismatch While Checking Service Description
				ELSIF udiStatus2 = 2727 THEN
					udiStatus2	:= 10087;	//MachineId Missing While Checking Service Description
				ELSIF udiStatus2 = 2728 THEN
					udiStatus2	:= 10088;	//LandId Out Of Range While Checking Service Description
				ELSIF udiStatus2 = 2729 THEN
					udiStatus2	:= 10089;	//LandId Missing While Checking Service Description
				ELSIF udiStatus2 = 2730 THEN
					udiStatus2	:= 10090;	//Version Missing While Checking Service Description
				ELSIF udiStatus2 = 2731 THEN
					udiStatus2	:= 10091;	//SupportedFeatures Missing While Checking Service Description
				END_IF

				fHermesAddOneMsgSend(ADR(a_eMsgSend) , ADR(udiMsgSendBffr) , HermesMsgTypeNotification);

				tyNotificationSnd.tyAvl.bSeverity			:= TRUE;
				tyNotificationSnd.tyAvl.bNotificationCode	:= TRUE;
				tyNotificationSnd.tyAvl.bDescription		:= TRUE;
				tyNotificationSnd.tyData.eSeverity			:= HermesSeverityFatalError;
				tyNotificationSnd.tyData.iNotificationCode	:= UDINT_TO_INT(udiStatus2);
				tyNotificationSnd.tyData.sDescription		:= a_tyAlmText[udiStatus2].sAlmText;

			END_IF
		END_IF

		IF tyMsgTypeRcv.bNotification = TRUE THEN
			udiStatus2	:= fHermesChkParamN(tyNotificationRcv);

			IF udiStatus2 <> 0 THEN
				eStatus2	:= Error;

				IF udiStatus2 = 2732 THEN
					udiStatus2	:= 10092;	//NotificationCode Out Of Range While Checking Notification
				ELSIF udiStatus2 = 2733 THEN
					udiStatus2	:= 10093;	//NotificationCode Missing While Checking Notification
				ELSIF udiStatus2 = 2734 THEN
					udiStatus2	:= 10094;	//Severity Missing While Checking Notification
				ELSIF udiStatus2 = 2735 THEN
					udiStatus2	:= 10095;	//Description Missing While Checking Notification
				END_IF

				fHermesAddOneMsgSend(ADR(a_eMsgSend) , ADR(udiMsgSendBffr) , HermesMsgTypeNotification);

				tyNotificationSnd.tyAvl.bSeverity			:= TRUE;
				tyNotificationSnd.tyAvl.bNotificationCode	:= TRUE;
				tyNotificationSnd.tyAvl.bDescription		:= TRUE;
				tyNotificationSnd.tyData.eSeverity			:= HermesSeverityFatalError;
				tyNotificationSnd.tyData.iNotificationCode	:= UDINT_TO_INT(udiStatus2);
				tyNotificationSnd.tyData.sDescription		:= a_tyAlmText[udiStatus2].sAlmText;

			END_IF
		END_IF

		IF tyMsgTypeRcv.bMachineReady = TRUE THEN
			udiStatus2	:= fHermesChkParamMR(tyMachineReady);

			IF udiStatus2 <> 0 THEN
				eStatus2	:= Error;

				IF udiStatus2 = 2740 THEN
					udiStatus2	:= 10098;	//FailedBoard Missing While Checking Machine Ready
				END_IF

				fHermesAddOneMsgSend(ADR(a_eMsgSend) , ADR(udiMsgSendBffr) , HermesMsgTypeNotification);

				tyNotificationSnd.tyAvl.bSeverity			:= TRUE;
				tyNotificationSnd.tyAvl.bNotificationCode	:= TRUE;
				tyNotificationSnd.tyAvl.bDescription		:= TRUE;
				tyNotificationSnd.tyData.eSeverity			:= HermesSeverityError;
				tyNotificationSnd.tyData.iNotificationCode	:= UDINT_TO_INT(udiStatus2);
				tyNotificationSnd.tyData.sDescription		:= a_tyAlmText[udiStatus2].sAlmText;

			END_IF
		END_IF

		IF tyMsgTypeRcv.bStartTransport = TRUE THEN
			udiStatus2	:= fHermesChkParamSAT(tyStartTransport);

			IF udiStatus2 <> 0 THEN
				eStatus2	:= Error;

				IF udiStatus2 = 2745 THEN
					udiStatus2	:= 10101;	//BoardId Missing While Checking Start Transport
				END_IF

				fHermesAddOneMsgSend(ADR(a_eMsgSend) , ADR(udiMsgSendBffr) , HermesMsgTypeNotification);

				tyNotificationSnd.tyAvl.bSeverity			:= TRUE;
				tyNotificationSnd.tyAvl.bNotificationCode	:= TRUE;
				tyNotificationSnd.tyAvl.bDescription		:= TRUE;
				tyNotificationSnd.tyData.eSeverity			:= HermesSeverityError;
				tyNotificationSnd.tyData.iNotificationCode	:= UDINT_TO_INT(udiStatus2);
				tyNotificationSnd.tyData.sDescription		:= a_tyAlmText[udiStatus2].sAlmText;

			END_IF
		END_IF

		IF tyMsgTypeRcv.bStopTransport = TRUE THEN
			udiStatus2	:= fHermesChkParamSOT(tyStopTransport);

			IF udiStatus2 <> 0 THEN
				eStatus2	:= Error;

				IF udiStatus2 = 2742 THEN
					udiStatus2	:= 10099;	//TransferState Missing While Checking Stop Transport
				ELSIF udiStatus2 = 2743 THEN
					udiStatus2	:= 10100;	//BoardId Missing While Checking Stop Transport
				END_IF

				fHermesAddOneMsgSend(ADR(a_eMsgSend) , ADR(udiMsgSendBffr) , HermesMsgTypeNotification);

				tyNotificationSnd.tyAvl.bSeverity			:= TRUE;
				tyNotificationSnd.tyAvl.bNotificationCode	:= TRUE;
				tyNotificationSnd.tyAvl.bDescription		:= TRUE;
				tyNotificationSnd.tyData.eSeverity			:= HermesSeverityError;
				tyNotificationSnd.tyData.iNotificationCode	:= UDINT_TO_INT(udiStatus2);
				tyNotificationSnd.tyData.sDescription		:= a_tyAlmText[udiStatus2].sAlmText;

			END_IF
		END_IF

		IF tyServiceDescriptionRcv.tyAvl.tySupportedFeatures.bFeatureQueryBoardInfo = TRUE AND p_tyParam.bFeatureSendBoardInfo THEN
			IF tyMsgTypeRcv.bQueryBoardInfo = TRUE THEN
				udiStatus2	:= fHermesChkParamQBI(tyQueryBoardInfo);

				IF udiStatus2 <> 0 THEN
					eStatus2	:= Error;

					IF udiStatus2 = 2766 THEN
						udiStatus2	:= 10102;	//Barcode Missing While Checking Query Board Info
					END_IF

					fHermesAddOneMsgSend(ADR(a_eMsgSend) , ADR(udiMsgSendBffr) , HermesMsgTypeNotification);

					tyNotificationSnd.tyAvl.bSeverity			:= TRUE;
					tyNotificationSnd.tyAvl.bNotificationCode	:= TRUE;
					tyNotificationSnd.tyAvl.bDescription		:= TRUE;
					tyNotificationSnd.tyData.eSeverity			:= HermesSeverityError;
					tyNotificationSnd.tyData.iNotificationCode	:= UDINT_TO_INT(udiStatus2);
					tyNotificationSnd.tyData.sDescription		:= a_tyAlmText[udiStatus2].sAlmText;

		        	tyMsgTypeRcv.bQueryBoardInfo := FALSE; //reset, else will latching
				END_IF
			END_IF
		END_IF

		IF tyMsgTypeRcv.bCommand = TRUE THEN
			udiStatus2 := fHermesChkParamCommand(tyCommandRcv);

			IF udiStatus2 <> 0 THEN
				eStatus2	:= Error;

				//				IF udiStatus2 = 2764 THEN
				//					udiStatus2	:= 10102;	//FailedBoard Missing While Checking Board Forecast
				//
				//				ELSIF udiStatus2 = 2765 THEN
				//					udiStatus2	:= 10103;	//FlippedBoard Missing While Checking Board Forecast
				//				END_IF

				fHermesAddOneMsgSend(ADR(a_eMsgSend) , ADR(udiMsgSendBffr) , HermesMsgTypeNotification);

				tyNotificationSnd.tyAvl.bSeverity			:= TRUE;
				tyNotificationSnd.tyAvl.bNotificationCode	:= TRUE;
				tyNotificationSnd.tyAvl.bDescription		:= TRUE;
				tyNotificationSnd.tyData.eSeverity			:= HermesSeverityError;
				tyNotificationSnd.tyData.iNotificationCode	:= UDINT_TO_INT(udiStatus2);
				tyNotificationSnd.tyData.sDescription		:= a_tyAlmText[udiStatus2].sAlmText;

			END_IF

		END_IF
	END_IF

END_ACTION
```

#### Act_Background_BoardForecast.st - Do Not Change!!!
```iecst
(** 2023-08-01 **)
ACTION Act_Background_BoardForecast:

	bFeatureBoardForecast := (p_tyParam.bFeatureBoardForecast = TRUE) AND (tyServiceDescriptionRcv.tyAvl.tySupportedFeatures.bFeatureBoardForecast = TRUE) (*AND bHandshakeDone*) ;

	IF NOT(bFeatureBoardForecast) THEN
		bNewChangeOver := FALSE;
		bSendBFNoID	   := FALSE;
		bSendBFId	   := FALSE;
		bBFIdSent	   := FALSE;
		bSndReverseBF  :=  FALSE;
		tyInfoData.sProgNm		:= '';
		tyInfoData.udiCode		:= 0;
		tyInfoData.eSeverity	:= AlmSeverityNA;
		tyInfoData.sAlmMsg		:= '';
	ELSE
		bSndReverseBF := EDGEPOS(p_usiUSHermesReverseDSSendBFId <> 0);

		fbTimerRstBFId(IN:= bSendBFId AND bBFIdSent
		AND NOT(bRstSendBFId) AND tyInfoData.udiCode= 10999
		AND bDSRdy
		,PT := T#1000s); //start counting when received mismatch Machine ready

		IF bRstSendBFId OR fbTimerRstBFId.Q
			OR EDGEPOS(bAllZoneEmpty AND p_bConvInitDone)  THEN //Reset BoardForecast width id
			bRstSendBFId := FALSE;
			bSendBFId := FALSE;
			bBFIdSent := FALSE;
		ELSIF fbTimerRstBFId.IN THEN
			sRstTim 				:= REAL_TO_STRING(TIME_TO_REAL(fbTimerRstBFId.PT-fbTimerRstBFId.ET)/1000.0);
			tyInfoData.sAlmMsg		:= CONCAT(sInfoMcRdyMsg,CONCAT(sRstTim,'(seconds)'));
		END_IF

		IF EDGEPOS(bNewProduct) OR EDGEPOS(bNewWidth) THEN  //Trigger BFID
			bNewChangeOver := TRUE;
			bBFIdSent := FALSE; //To resend BF-ID
		END_IF

		IF bNewChangeOver AND bAllZoneEmpty AND p_bConvInitDone THEN
			bNewChangeOver:= FALSE;
			bSendBFId	  := TRUE; //reset when find mactch machine ready
		END_IF

		IF bSendBFId = FALSE AND bBFIdSent = FALSE THEN //reset notification
			tyInfoData.sProgNm		:= '';
			tyInfoData.udiCode		:= 0;
			tyInfoData.eSeverity	:= AlmSeverityNA;
			tyInfoData.sAlmMsg		:= '';
		END_IF

		IF bSendBFId = FALSE   THEN  	//Trigger BF No Id
			bSendBFNoID	:= FALSE;
			IF bFirstZoneHaveBoard AND NOT(bFirstZoneEndSen) THEN //Zone 1 PCB_In and have Board
				bSendBFNoID	:= TRUE;
			ELSIF bSndReverseBF THEN // EDGEPOS(bSndReverseBF) OR EDGENEG(bSndReverseBF) THEN //Reverse route
				bSendBFNoID	:= TRUE; //EDGEPOS send Brd id , EDGENEG send empty brd id
			END_IF
		END_IF

	END_IF

END_ACTION
```

#### Act_Background_SendBoardInfo.st - Do Not Change!!!
```iecst
(** 2021-08-01 **)
ACTION Act_Background_SendBoardInfo:
	// back-up to array when finished transport

	IF NOT(tyServiceDescriptionRcv.tyAvl.tySupportedFeatures.bFeatureQueryBoardInfo = TRUE AND p_tyParam.bFeatureSendBoardInfo AND bHandshakeDone) THEN
		bSearchTop := FALSE;
		bSearchBottom := FALSE;
		siTopBarcodeIdx := -1;
		siBottomBarcodeIdx := -1;
		siFoundIdx	:= -1;
	ELSE
		IF eStatus2  <> Error THEN
			//search
			IF tyMsgTypeRcv.bQueryBoardInfo THEN
				tyMsgTypeRcv.bQueryBoardInfo := FALSE;

				bSearchTop := tyQueryBoardInfo.tyData.sTopBarcode <> '';
				bSearchBottom := tyQueryBoardInfo.tyData.sBottomBarcode <> '';

				siTopBarcodeIdx := -1;
				siBottomBarcodeIdx := -1;
				FOR siSearhIdx := 0 TO SIZEOF(a_tyBoardDepartedInfo)/SIZEOF(a_tyBoardDepartedInfo[0])-1 DO
					IF bSearchTop THEN
						IF memcmp(ADR(tyQueryBoardInfo.tyData.sTopBarcode),
							ADR(a_tyBoardDepartedInfo[0].tyData.sTopBarcode)+siSearhIdx*SIZEOF(a_tyBoardDepartedInfo[0]),
							SIZEOF(tyQueryBoardInfo.tyData.sTopBarcode)) = 0 THEN
								siTopBarcodeIdx	:= siSearhIdx;
						END_IF
					END_IF

					IF bSearchBottom THEN
						IF memcmp(ADR(tyQueryBoardInfo.tyData.sBottomBarcode),
							ADR(a_tyBoardDepartedInfo[0].tyData.sBottomBarcode)+siSearhIdx*SIZEOF(a_tyBoardDepartedInfo[0]),
							SIZEOF(tyQueryBoardInfo.tyData.sBottomBarcode)) = 0 THEN
								siBottomBarcodeIdx := siSearhIdx;
						END_IF
					END_IF

					IF (NOT(bSearchTop) OR ( bSearchTop AND siTopBarcodeIdx <> -1 ) ) AND
						(NOT(bSearchBottom) OR( bSearchBottom AND siBottomBarcodeIdx <> -1 ))THEN
						EXIT;
					END_IF
				END_FOR

				bCompleteSearch 	:= NOT(bSearchTop AND siTopBarcodeIdx =  -1)
										AND NOT(bSearchBottom AND siBottomBarcodeIdx = -1)
										AND NOT(bSearchTop AND bSearchBottom AND siTopBarcodeIdx <> siBottomBarcodeIdx );
				IF bCompleteSearch THEN
					IF siTopBarcodeIdx <> -1 THEN
						siFoundIdx := siTopBarcodeIdx;
					ELSIF siBottomBarcodeIdx <> -1 THEN
						siFoundIdx := siBottomBarcodeIdx;
					END_IF
					fHermesAddOneMsgSend(ADR(a_eMsgSend) , ADR(udiMsgSendBffr) , HermesMsgTypeSendBoardInfo);

					tySendBoardInfo.tyData.sBoardId                     := a_tyBoardDepartedInfo[siFoundIdx].tyData.sBoardId;
					tySendBoardInfo.tyData.sBoardIdCreatedBy            := a_tyBoardDepartedInfo[siFoundIdx].tyData.sBoardIdCreatedBy;
					tySendBoardInfo.tyData.eFailedBoard 		    	:= a_tyBoardDepartedInfo[siFoundIdx].tyData.eFailedBoard;
					tySendBoardInfo.tyData.sProductTypeId 			    := a_tyBoardDepartedInfo[siFoundIdx].tyData.sProductTypeId;	 //current recipe0 name
					tySendBoardInfo.tyData.eFlippedBoard 		    	:= a_tyBoardDepartedInfo[siFoundIdx].tyData.eFlippedBoard;
					tySendBoardInfo.tyData.sTopBarcode 		        	:= a_tyBoardDepartedInfo[siFoundIdx].tyData.sTopBarcode;
					tySendBoardInfo.tyData.sBottomBarcode 		    	:= a_tyBoardDepartedInfo[siFoundIdx].tyData.sBottomBarcode;
					tySendBoardInfo.tyData.rLength 			        	:= a_tyBoardDepartedInfo[siFoundIdx].tyData.rLength;
					tySendBoardInfo.tyData.rWidth 			        	:= a_tyBoardDepartedInfo[siFoundIdx].tyData.rWidth;	//current recipe 0 width
					tySendBoardInfo.tyData.rThickness 		        	:= a_tyBoardDepartedInfo[siFoundIdx].tyData.rThickness;
					tySendBoardInfo.tyData.rTopClearanceHeight 	    	:= a_tyBoardDepartedInfo[siFoundIdx].tyData.rTopClearanceHeight;
					tySendBoardInfo.tyData.rBottomClearanceHeight 	    := a_tyBoardDepartedInfo[siFoundIdx].tyData.rBottomClearanceHeight;
					tySendBoardInfo.tyData.rWeight 			        	:= a_tyBoardDepartedInfo[siFoundIdx].tyData.rWeight;
					tySendBoardInfo.tyData.sWorkOrderId 		    	:= a_tyBoardDepartedInfo[siFoundIdx].tyData.sWorkOrderId;

					tySendBoardInfo.tyAvl.bBoardId 				        := tySendBoardInfo.tyData.sBoardId <> '';
					tySendBoardInfo.tyAvl.bBoardIdCreatedBy 	        := tySendBoardInfo.tyData.sBoardIdCreatedBy <> '';
					tySendBoardInfo.tyAvl.bFailedBoard 			        := TRUE;
					tySendBoardInfo.tyAvl.bProductTypeId 		    	:= tySendBoardInfo.tyData.sProductTypeId <> '';
					tySendBoardInfo.tyAvl.bFlippedBoard 		        := TRUE;
					tySendBoardInfo.tyAvl.bTopBarcode 		    	    := tySendBoardInfo.tyData.sTopBarcode <> '';
					tySendBoardInfo.tyAvl.bBottomBarcode 		    	:= tySendBoardInfo.tyData.sBottomBarcode <> '';
					tySendBoardInfo.tyAvl.bLength 			        	:= tySendBoardInfo.tyData.rLength <> 0;
					tySendBoardInfo.tyAvl.bWidth						:= tySendBoardInfo.tyData.rWidth <> 0;
					tySendBoardInfo.tyAvl.bThickness 		        	:= tySendBoardInfo.tyData.rThickness <> 0;
					tySendBoardInfo.tyAvl.bTopClearanceHeight 	    	:= tySendBoardInfo.tyData.rTopClearanceHeight <> 0;
					tySendBoardInfo.tyAvl.bBottomClearanceHeight 	    := tySendBoardInfo.tyData.rBottomClearanceHeight <> 0;
					tySendBoardInfo.tyAvl.bWeight 			        	:= tySendBoardInfo.tyData.rWeight <> 0;
					tySendBoardInfo.tyAvl.bWorkOrderId 		        	:= tySendBoardInfo.tyData.sWorkOrderId <> '';

				ELSE
					fHermesAddOneMsgSend(ADR(a_eMsgSend) , ADR(udiMsgSendBffr) , HermesMsgTypeSendBoardInfo);

					tySendBoardInfo.tyData.sBoardId                     := '';
					tySendBoardInfo.tyData.sBoardIdCreatedBy            := '';
					tySendBoardInfo.tyData.eFailedBoard 		    	:= HermesUnknownBoard;
					tySendBoardInfo.tyData.sProductTypeId 			    := '';
					tySendBoardInfo.tyData.eFlippedBoard 		    	:= HermesFlippedBoardUnknownSide;
					tySendBoardInfo.tyData.sTopBarcode 		        	:= tyQueryBoardInfo.tyData.sTopBarcode;
					tySendBoardInfo.tyData.sBottomBarcode 		    	:= tyQueryBoardInfo.tyData.sBottomBarcode;
					tySendBoardInfo.tyData.rLength 			        	:= 0;
					tySendBoardInfo.tyData.rWidth 			        	:= 0;
					tySendBoardInfo.tyData.rThickness 		        	:= 0;
					tySendBoardInfo.tyData.rTopClearanceHeight 	    	:= 0;
					tySendBoardInfo.tyData.rBottomClearanceHeight 	    := 0;
					tySendBoardInfo.tyData.rWeight 			        	:= 0;
					tySendBoardInfo.tyData.sWorkOrderId 		    	:= '';
					tySendBoardInfo.tyData.sBatchId      		    	:= '';

					tySendBoardInfo.tyAvl.bBoardId 				        := tySendBoardInfo.tyData.sBoardId <> '';
					tySendBoardInfo.tyAvl.bBoardIdCreatedBy 	        := tySendBoardInfo.tyData.sBoardIdCreatedBy <> '';
					tySendBoardInfo.tyAvl.bFailedBoard 			        := FALSE; //no need send
					tySendBoardInfo.tyAvl.bProductTypeId 		    	:= tySendBoardInfo.tyData.sProductTypeId <> '';
					tySendBoardInfo.tyAvl.bFlippedBoard 	    	    := FALSE; //no need send
					tySendBoardInfo.tyAvl.bTopBarcode 		        	:= tySendBoardInfo.tyData.sTopBarcode <> '';
					tySendBoardInfo.tyAvl.bBottomBarcode 	    		:= tySendBoardInfo.tyData.sBottomBarcode <> '';
					tySendBoardInfo.tyAvl.bLength 			        	:= tySendBoardInfo.tyData.rLength <> 0;
					tySendBoardInfo.tyAvl.bWidth 			        	:= tySendBoardInfo.tyData.rWidth <> 0;
					tySendBoardInfo.tyAvl.bThickness 		        	:= tySendBoardInfo.tyData.rThickness <> 0;
					tySendBoardInfo.tyAvl.bTopClearanceHeight 	    	:= tySendBoardInfo.tyData.rTopClearanceHeight <> 0;
					tySendBoardInfo.tyAvl.bBottomClearanceHeight     	:= tySendBoardInfo.tyData.rBottomClearanceHeight <> 0;
					tySendBoardInfo.tyAvl.bWeight 			        	:= tySendBoardInfo.tyData.rWeight <> 0;
					tySendBoardInfo.tyAvl.bWorkOrderId 		        	:= tySendBoardInfo.tyData.sWorkOrderId <> '';
					tySendBoardInfo.tyAvl.bBatchId 		            	:= tySendBoardInfo.tyData.sBatchId <> '';

				END_IF

			END_IF
		END_IF
	END_IF
	//search

END_ACTION
```

#### Act_Background_Route.st - Do Not Change!!!
```iecst
(** 2021-08-01 **)
ACTION Act_Background_Route:

	//DS Routing Function

	//same lane same interface
	//reverse output

	IF NOT(p_bProcessRouteEn) THEN

		bTriggerRouteReversal := FALSE;
	ELSE
		//decision making re-route the route number
		IF EDGEPOS(tyBoardAvailableRcv.tyAvl.bFlippedBoard  AND tyBoardAvailableRcv.tyData.eFlippedBoard = HermesFlippedBoardTopSideUp) THEN
			bTriggerRouteReversal := TRUE;
		END_IF

		IF p_bReturnRoute AND bTriggerRouteReversal  THEN //Process machine as upstream
			bTriggerRouteReversal := FALSE;
			iRoute := 990;
		END_IF

	END_IF

	//revese route, send
	IF NOT(p_bReverseSentRoute) THEN
		bSwitchtoReverseSend := FALSE;
	ELSE
		IF bReverseDSSndBfWBrdID = FALSE AND tyMsgTypeRcv.bMachineReady AND tyBoardForecastSnd.tyData.sBoardId = tyMachineReady.tyData.sBoardId THEN
			bSwitchtoReverseSend := TRUE;
//			IF p_bUSHermesProcessRouteTrigger THEN
//				iRoute := 990;
//			ELSE
//				iRoute := 0;
//			END_IF
		ELSIF bReverseDSSndBfWBrdID = TRUE
			AND ( EDGEPOS(tyMsgTypeRcv.bStopTransport AND tyStopTransport.tyData.eTransferState = HermesTransferStateComplete )
			)THEN
			bSwitchtoReverseSend := FALSE;
		END_IF

		fbRstReverseSndGate(IN:= bSwitchtoReverseSend);
		bNotifyRstReverseSndGate := fbRstReverseSndGate.Q;

		//feedback
		//bDSHermesRcvReverseUSMcRdy :=
		bReverseRcvBlkDS :=  NOT(bSwitchtoReverseSend);
	END_IF

END_ACTION
```
